METHOD setCirclePlane : BOOL //Return value = TRUE if executed succesful
VAR_INPUT
	X														: LREAL := 0.0;
	Y														: LREAL := 0.0;
	Z														: LREAL := 0.0;
	Q1														: LREAL := 0.0;
	Q2														: LREAL := 0.0;
	Q3														: LREAL := 0.0;
	Q4														: LREAL := 0.0;
	Q5														: LREAL := 0.0;
	Velo													: LREAL; 	// mm/s 
	AccurateStop											: BOOL := FALSE;
	Clockwise												: BOOL := TRUE;
	Plane													: E_NciGeoPlane := E_NciGeoPlaneXY;
	CenterX													: LREAL := 0.0;
	CenterY													: LREAL := 0.0;
	CenterZ													: LREAL := 0.0;
END_VAR
	(* NCI GeoCirclePlane schreiben									*)
	(*********************************************************)

(* Zielpos. in Tabelle schreiben ************************************************************)
	BlockCount 												:= BlockCount + 1;
	TblTemplate.GeoCirclePlane.nDisplayIndex := LastBlockNo := SEL(BlockNo = 0, BlockNo, TableNumber * OffsetFactorTblNumber + BlockCount);
	TblTemplate.GeoCirclePlane.fEndPosX						:= X;
	TblTemplate.GeoCirclePlane.fEndPosY						:= Y;
	TblTemplate.GeoCirclePlane.fEndPosZ						:= Z;
	TblTemplate.GeoCirclePlane.fEndPosQ1					:= Q1;
	TblTemplate.GeoCirclePlane.fEndPosQ2					:= Q2;
	TblTemplate.GeoCirclePlane.fEndPosQ3					:= Q3;
	TblTemplate.GeoCirclePlane.fEndPosQ4					:= Q4;
	TblTemplate.GeoCirclePlane.fEndPosQ5					:= Q5;
	TblTemplate.GeoCirclePlane.fVelo						:= Velo;
	TblTemplate.GeoCirclePlane.bAccurateStop				:= AccurateStop;
	TblTemplate.GeoCirclePlane.bClockwise					:= Clockwise;
	TblTemplate.GeoCirclePlane.nPlane						:= Plane;
	TblTemplate.GeoCirclePlane.fCenterX						:= CenterX;
	TblTemplate.GeoCirclePlane.fCenterY						:= CenterY;
	TblTemplate.GeoCirclePlane.fCenterZ						:= CenterZ;
                                                        	
	TblTemplate.InsertGeoCirclePlane(Table:= Table);    	
	Error													:= TblTemplate.Error;
	ErrorId													:= TblTemplate.ErrorId;
	ErrorText												:= TblTemplate.ErrorText;
	FilledRows												:= TblTemplate.FilledRows;

	SetCirclePlane											:= NOT Error;
(***************************************************************************)
END_METHOD

METHOD setCoordinateSystem : BOOL //Return value = TRUE if executed succesful
VAR_INPUT
	/// UCS ObjectID 
	ObjectId												: UDINT := 0;
END_VAR
(* NCI UserKos schreiben															*)
(************************************************************************************)

(* User Koordinatensystem schreiben ************************************************************)
	BlockCount 												:= BlockCount + 1;
	TblTemplate.SetCoordinateSystem.nDisplayIndex := LastBlockNo := SEL(BlockNo = 0, BlockNo, TableNumber * OffsetFactorTblNumber + BlockCount);
	TblTemplate.SetCoordinateSystem.nObjectId				:= ObjectId;

	TblTemplate.InsertSetCoordinateSystem(Table:= Table);
	Error													:= TblTemplate.Error;
	ErrorId													:= TblTemplate.ErrorId;
	ErrorText												:= TblTemplate.ErrorText;
	FilledRows												:= TblTemplate.FilledRows;
	
	SetCoordinateSystem										:= not Error;
(*************************************************************************************)
END_METHOD

METHOD setDynOverride : BOOL //Return value = TRUE if executed succesful
VAR_INPUT
	/// UCS ObjectID 
	Value													: lreal := 0; //0.0-100.0%
END_VAR
(* NCI Oevrride schreiben											*)
(********************************************************************)

(* insert override **************************************************)
	(* apapt override *)
	BlockCount 												:= BlockCount + 1;
	TblTemplate.DynOverride.nDisplayIndex := LastBlockNo 		:= SEL(BlockNo = 0, BlockNo, TableNumber * OffsetFactorTblNumber + BlockCount);
	TblTemplate.DynOverride.fDynOvr								:= 0.01 * Value;

	TblTemplate.InsertDynOverride(Table:= Table);
	Error													:= TblTemplate.Error;
	ErrorId													:= TblTemplate.ErrorId;
	ErrorText												:= TblTemplate.ErrorText;
	FilledRows												:= TblTemplate.FilledRows;
	
	SetDynOverride											:= not Error;
(*************************************************************************************)
END_METHOD

METHOD setGeoBezier3 : booL //Return value = TRUE if executed succesful
VAR_INPUT
     ControlPoint1X											: LREAL;
     ControlPoint1Y											: LREAL;
     ControlPoint1Z											: LREAL;
     ControlPoint2X											: LREAL;
     ControlPoint2Y											: LREAL;
     ControlPoint2Z											: LREAL;
     EndPosX												: LREAL;
     EndPosY												: LREAL;
     EndPosZ												: LREAL;
     EndPosQ1												: LREAL;
     EndPosQ2												: LREAL;
     EndPosQ3												: LREAL;
     EndPosQ4												: LREAL;
     EndPosQ5												: LREAL;
     Velo													: LREAL;
     AccurateStop											: BOOL; (* VeloEnd := 0 *)
END_VAR
	(* NCI SetGeoBezier3 schreiben						*)
	(*********************************************************)

(* Zielpos. in Tabelle schreiben ************************************************************)
	BlockCount 												:= BlockCount + 1;
	TblTemplate.GeoBezier3.nDisplayIndex := LastBlockNo := SEL(BlockNo = 0, BlockNo, TableNumber * OffsetFactorTblNumber + BlockCount);

    TblTemplate.GeoBezier3.fControlPoint1X					:= ControlPoint1X;
    TblTemplate.GeoBezier3.fControlPoint1Y					:= ControlPoint1Y;
    TblTemplate.GeoBezier3.fControlPoint1Z					:= ControlPoint1Z;
    TblTemplate.GeoBezier3.fControlPoint2X					:= ControlPoint2X;
    TblTemplate.GeoBezier3.fControlPoint2Y					:= ControlPoint2Y;
    TblTemplate.GeoBezier3.fControlPoint2Z					:= ControlPoint2Z;
    TblTemplate.GeoBezier3.fEndPosX							:= EndPosX;
    TblTemplate.GeoBezier3.fEndPosY							:= EndPosY;
    TblTemplate.GeoBezier3.fEndPosZ							:= EndPosZ;
    TblTemplate.GeoBezier3.fEndPosQ1						:= EndPosQ1;
    TblTemplate.GeoBezier3.fEndPosQ2						:= EndPosQ2;
    TblTemplate.GeoBezier3.fEndPosQ3						:= EndPosQ3;
    TblTemplate.GeoBezier3.fEndPosQ4						:= EndPosQ4;
    TblTemplate.GeoBezier3.fEndPosQ5						:= EndPosQ5;
    TblTemplate.GeoBezier3.fVelo							:= Velo;
    TblTemplate.GeoBezier3.bAccurateStop					:= AccurateStop  ;                            	
	
	TblTemplate.InsertGeoBezier3(Table:= Table);    	
	Error													:= TblTemplate.Error;
	ErrorId													:= TblTemplate.ErrorId;
	ErrorText												:= TblTemplate.ErrorText;
	FilledRows												:= TblTemplate.FilledRows;

	SetGeoBezier3											:= NOT Error;
(***************************************************************************)
END_METHOD

METHOD setGeoBezier5 : booL //Return value = TRUE if executed succesful
VAR_INPUT
     ControlPoint1X											: LREAL;
     ControlPoint1Y											: LREAL;
     ControlPoint1Z											: LREAL;
     ControlPoint2X											: LREAL;
     ControlPoint2Y											: LREAL;
     ControlPoint2Z											: LREAL;
     ControlPoint3X											: LREAL;
     ControlPoint3Y											: LREAL;
     ControlPoint3Z											: LREAL;
     ControlPoint4X											: LREAL;
     ControlPoint4Y											: LREAL;
     ControlPoint4Z											: LREAL;
     EndPosX												: LREAL;
     EndPosY												: LREAL;
     EndPosZ												: LREAL;
     EndPosQ1												: LREAL;
     EndPosQ2												: LREAL;
     EndPosQ3												: LREAL;
     EndPosQ4												: LREAL;
     EndPosQ5												: LREAL;
     Velo													: LREAL;
     AccurateStop											: BOOL; (* VeloEnd := 0 *)
END_VAR
	(* NCI SetGeoBezier5 schreiben						*)
	(*********************************************************)

(* Zielpos. in Tabelle schreiben ************************************************************)
	BlockCount 												:= BlockCount + 1;
	TblTemplate.GeoBezier5.nDisplayIndex := LastBlockNo := SEL(BlockNo = 0, BlockNo, TableNumber * OffsetFactorTblNumber + BlockCount);

    TblTemplate.GeoBezier5.fControlPoint1X					:= ControlPoint1X;
    TblTemplate.GeoBezier5.fControlPoint1Y					:= ControlPoint1Y;
    TblTemplate.GeoBezier5.fControlPoint1Z					:= ControlPoint1Z;
    TblTemplate.GeoBezier5.fControlPoint2X					:= ControlPoint2X;
    TblTemplate.GeoBezier5.fControlPoint2Y					:= ControlPoint2Y;
    TblTemplate.GeoBezier5.fControlPoint2Z					:= ControlPoint2Z;
    TblTemplate.GeoBezier5.fControlPoint3X					:= ControlPoint3X;
    TblTemplate.GeoBezier5.fControlPoint3Y					:= ControlPoint3Y;
    TblTemplate.GeoBezier5.fControlPoint3Z					:= ControlPoint3Z;
    TblTemplate.GeoBezier5.fControlPoint4X					:= ControlPoint4X;
    TblTemplate.GeoBezier5.fControlPoint4Y					:= ControlPoint4Y;
    TblTemplate.GeoBezier5.fControlPoint4Z					:= ControlPoint4Z;
    TblTemplate.GeoBezier5.fEndPosX							:= EndPosX;
    TblTemplate.GeoBezier5.fEndPosY							:= EndPosY;
    TblTemplate.GeoBezier5.fEndPosZ							:= EndPosZ;
    TblTemplate.GeoBezier5.fEndPosQ1						:= EndPosQ1;
    TblTemplate.GeoBezier5.fEndPosQ2						:= EndPosQ2;
    TblTemplate.GeoBezier5.fEndPosQ3						:= EndPosQ3;
    TblTemplate.GeoBezier5.fEndPosQ4						:= EndPosQ4;
    TblTemplate.GeoBezier5.fEndPosQ5						:= EndPosQ5;
    TblTemplate.GeoBezier5.fVelo							:= Velo;
    TblTemplate.GeoBezier5.bAccurateStop					:= AccurateStop  ;                            	
	
	TblTemplate.InsertGeoBezier5(Table:= Table);    	
	Error													:= TblTemplate.Error;
	ErrorId													:= TblTemplate.ErrorId;
	ErrorText												:= TblTemplate.ErrorText;
	FilledRows												:= TblTemplate.FilledRows;

	SetGeoBezier5											:= NOT Error;
(***************************************************************************)
END_METHOD

METHOD setGeoLine : BOOL //Return value = TRUE if executed succesful
VAR_INPUT
	X														: LREAL := 0.0;
	Y														: LREAL := 0.0;
	Z														: LREAL := 0.0;
	Q1														: LREAL := 0.0;
	Q2														: LREAL := 0.0;
	Q3														: LREAL := 0.0;
	Q4														: LREAL := 0.0;
	Q5														: LREAL := 0.0;
	Velo													: LREAL; 	// mm/s 
	AccurateStop											: BOOL := FALSE;
END_VAR
(* writing NCI GeoLine 									*)
(********************************************************)

(***************************************************************************)
	BlockCount 												:= BlockCount + 1;
	TblTemplate.GeoLine.nDisplayIndex := LastBlockNo 		:= SEL(BlockNo = 0, BlockNo, TableNumber * OffsetFactorTblNumber + BlockCount);
	TblTemplate.GeoLine.fEndPosX							:= X;
	TblTemplate.GeoLine.fEndPosY							:= Y;
	TblTemplate.GeoLine.fEndPosZ							:= Z;
	TblTemplate.GeoLine.fEndPosQ1							:= Q1 ;
	TblTemplate.GeoLine.fEndPosQ2							:= Q2;
	TblTemplate.GeoLine.fEndPosQ3							:= Q3;
	TblTemplate.GeoLine.fEndPosQ4							:= Q4;
	TblTemplate.GeoLine.fEndPosQ5							:= Q5;
	TblTemplate.GeoLine.fVelo								:= Velo;
	TblTemplate.GeoLine.bRapidTraverse						:= Velo = 0.0;
	TblTemplate.GeoLine.bAccurateStop						:= AccurateStop;
                                                        	
	TblTemplate.InsertGeoLine(Table:= Table);           	
	Error													:= TblTemplate.Error;
	ErrorId													:= TblTemplate.ErrorId;
	ErrorText												:= TblTemplate.ErrorText;
	FilledRows												:= TblTemplate.FilledRows;
	
	SetGeoLine												:= not Error;
(***************************************************************************)
END_METHOD

METHOD setGeoStart : BOOL //Return value = TRUE if executed succesful
VAR_INPUT
	X														: LREAL := 0.0;
	Y														: LREAL := 0.0;
	Z														: LREAL := 0.0;
	Q1														: LREAL := 0.0;
	Q2														: LREAL := 0.0;
	Q3														: LREAL := 0.0;
	Q4														: LREAL := 0.0;
	Q5														: LREAL := 0.0;
END_VAR
(* writing NCI GeoLine 									*)
(********************************************************)

(***************************************************************************)
	TblTemplate.GeoStart.fPosX								:= X;
	TblTemplate.GeoStart.fPosY								:= Y;
	TblTemplate.GeoStart.fPosZ								:= Z;
	TblTemplate.GeoStart.fPosQ1								:= Q1 ;
	TblTemplate.GeoStart.fPosQ2								:= Q2;
	TblTemplate.GeoStart.fPosQ3								:= Q3;
	TblTemplate.GeoStart.fPosQ4								:= Q4;
	TblTemplate.GeoStart.fPosQ5								:= Q5;
                                                        	
	TblTemplate.InsertGeoStart(Table:= Table);           	
	Error													:= TblTemplate.Error;
	ErrorId													:= TblTemplate.ErrorId;
	ErrorText												:= TblTemplate.ErrorText;
	FilledRows												:= TblTemplate.FilledRows;
	
	SetGeoStart												:= not Error;
(***************************************************************************)
END_METHOD

METHOD setHParam : booL //Return value = TRUE if executed succesful
VAR_INPUT
	HParam													: UDINT;
END_VAR
(* 														*)
(********************************************************)

(*************************************************************************************)
	BlockCount 												:= BlockCount + 1;
	TblTemplate.HParam.nDisplayIndex := LastBlockNo 		:= SEL(BlockNo = 0, BlockNo,  TableNumber * OffsetFactorTblNumber + BlockCount);
	TblTemplate.HParam.nHParam								:= HParam;
                                                        	
	TblTemplate.InsertHParam(Table:= Table);          	
	Error													:= TblTemplate.Error;
	ErrorId													:= TblTemplate.ErrorId;
	ErrorText												:= TblTemplate.ErrorText;
	FilledRows												:= TblTemplate.FilledRows;
	
	SetHParam												:= NOT Error;
(*************************************************************************************)
END_METHOD

METHOD setPathDynamics : BOOL //Return value = TRUE if executed succesful
VAR_INPUT
	Acc,Dec,Jerk											:	LREAL;
END_VAR
	(* NCI SetPathDynamics schreiben						*)
	(*********************************************************)

(* Zielpos. in Tabelle schreiben ************************************************************)
	BlockCount 												:= BlockCount + 1;
	TblTemplate.PathDynamics.nDisplayIndex := LastBlockNo := SEL(BlockNo = 0, BlockNo, TableNumber * OffsetFactorTblNumber + BlockCount);

	TblTemplate.PathDynamics.fDec							:= Dec;
	TblTemplate.PathDynamics.fJerk							:= Jerk;
	TblTemplate.PathDynamics.fAcc							:= Acc;
                                                        	
	TblTemplate.InsertPathDynamics(Table:= Table);    	
	Error													:= TblTemplate.Error;
	ErrorId													:= TblTemplate.ErrorId;
	ErrorText												:= TblTemplate.ErrorText;
	FilledRows												:= TblTemplate.FilledRows;

	SetPathDynamics											:= NOT Error;
(***************************************************************************)
END_METHOD

METHOD setSParam : bool //Return value = TRUE if executed succesful
VAR_INPUT
	SParam													: UINT;
END_VAR
(* 														*)
(********************************************************)

(*************************************************************************************)
	BlockCount 												:= BlockCount + 1;
	TblTemplate.SParam.nDisplayIndex := LastBlockNo 		:= SEL(BlockNo = 0, BlockNo,  TableNumber * OffsetFactorTblNumber + BlockCount);
	TblTemplate.SParam.nSParam								:= SParam;
                                                        	
	TblTemplate.InsertSParam(Table:= Table);          	
	Error													:= TblTemplate.Error;
	ErrorId													:= TblTemplate.ErrorId;
	ErrorText												:= TblTemplate.ErrorText;
	FilledRows												:= TblTemplate.FilledRows;
	
	SetSParam												:= NOT Error;
(*************************************************************************************)
END_METHOD

METHOD setTangFollowingDesc : booL //Return value = TRUE if executed succesful
VAR_INPUT
    TangOn													: BOOL;
    TangAxis												: E_NciAxesInGroup;  
    PathAxis1												: E_NciAxesInGroup; 
    PathAxis2												: E_NciAxesInGroup; 
    Offset													: LREAL; 
    CriticalAngle1											: LREAL;
    TfBehavior												: E_TangentialFollowingBehavior; 
END_VAR
	(* NCI SetTangFollowingDesc schreiben						*)
	(*********************************************************)

(* Zielpos. in Tabelle schreiben ************************************************************)
	BlockCount 												:= BlockCount + 1;
	LastBlockNo 											:= SEL(BlockNo = 0, BlockNo, TableNumber * OffsetFactorTblNumber + BlockCount);

    TblTemplate.TangentialFollowingDesc.bTangOn				:= TangOn;
    TblTemplate.TangentialFollowingDesc.nTangAxis			:= TangAxis;
    TblTemplate.TangentialFollowingDesc.nPathAxis1			:= PathAxis1;
    TblTemplate.TangentialFollowingDesc.nPathAxis2			:= PathAxis2;
    TblTemplate.TangentialFollowingDesc.fOffset				:= Offset;
    TblTemplate.TangentialFollowingDesc.fCriticalAngle1		:= CriticalAngle1;
    TblTemplate.TangentialFollowingDesc.nTfBehavior			:= TfBehavior;
                       	
	TblTemplate.InsertTangFollowingDesc(Table:= Table);    	
	Error													:= TblTemplate.Error;
	ErrorId													:= TblTemplate.ErrorId;
	ErrorText												:= TblTemplate.ErrorText;
	FilledRows												:= TblTemplate.FilledRows;

	SetTangFollowingDesc									:= NOT Error;
(***************************************************************************)
END_METHOD

METHOD setTParam : bool //Return value = TRUE if executed succesful
VAR_INPUT
	TParam													: UINT;
END_VAR
(* 														*)
(********************************************************)

(*************************************************************************************)
	BlockCount 												:= BlockCount + 1;
	TblTemplate.TParam.nDisplayIndex := LastBlockNo 		:= SEL(BlockNo = 0, BlockNo,  TableNumber * OffsetFactorTblNumber + BlockCount);
	TblTemplate.TParam.nTParam								:= TParam;
                                                        	
	TblTemplate.InsertTParam(Table:= Table);          	
	Error													:= TblTemplate.Error;
	ErrorId													:= TblTemplate.ErrorId;
	ErrorText												:= TblTemplate.ErrorText;
	FilledRows												:= TblTemplate.FilledRows;
	
	SetTParam												:= NOT Error;
(**************************************************************************)
END_METHOD

METHOD setVertexSmoothing : BOOL //Return value = TRUE if executed succesful
VAR_INPUT
	Radius													: LREAL := 0.0;
	VertSmType												: UDINT := 5;
	VertSmSubType											: UDINT := 3;
END_VAR
(* writing NCI Vertex smoothing 								*)
(****************************************************************)

(* writing into table	*****************************************)
	BlockCount 												:= BlockCount + 1;
	TblTemplate.VertexSmoothing.nDisplayIndex := LastBlockNo := SEL(BlockNo = 0, BlockNo, TableNumber * OffsetFactorTblNumber + BlockCount);
	TblTemplate.VertexSmoothing.nType						:= VertSmType;
	TblTemplate.VertexSmoothing.nSubtype					:= VertSmSubtype; (* 	1: constant radius tolerance
																					2: distance between Abstand intersectoin point and peal point
																					3: adaptiv raidus tolerance
																					*)
	TblTemplate.VertexSmoothing.fRadius						:= Radius; (* mm *)

	TblTemplate.InsertVertexSmoothing(Table:= Table);
	Error													:= TblTemplate.Error;
	ErrorId													:= TblTemplate.ErrorId;
	ErrorText												:= TblTemplate.ErrorText;
	FilledRows												:= TblTemplate.FilledRows;
	SetVertexSmoothing										:= not Error;
(*************************************************************************************)
END_METHOD

END_FUNCTION_BLOCK

// ---- POUs/Motion/TF511x-KIN/KinChannel.TcPOU
FUNCTION_BLOCK KinChannel EXTENDS KIN_REF
VAR_INPUT
	Admin													:	KinAdmin;
END_VAR
VAR_OUTPUT
END_VAR
VAR
END_VAR

(* Kinematic Ctrl 										*)
(********************************************************)

(* work IO ********************************************************************)
(*	IO(); *)
	
(****************************************************************************)
(* Kinematic group control													*)
(****************************************************************************)
	Admin(
		ResetTrig			:= ,
		Enable			:= ,
		Override		:= ,
		ItpChannelId	:= ,
		AxesList		:= ,
		rKINRef			:= THIS^,
		Busy			=> ,
		Done			=> ,
		Error			=> ,
		ErrorId			=> );
(****************************************************************************)

END_FUNCTION_BLOCK

// ---- POUs/Motion/TF50xx-NC/02_Options/Coupling/AxCamming.TcPOU
{attribute 'no_check'}
//Nc-axis camming (cam tabel) control
//based on Tc2_MC2_Camming library
FUNCTION_BLOCK AxCamming EXTENDS AxFbBase
VAR_OUTPUT CONSTANT
	FNC_CAM_OUT												:	INT := 0;
	FNC_CAM_IN												:	INT := 1;
END_VAR                     								
VAR_INPUT                   								
	Fnc														:	INT (FNC_CAM_OUT..FNC_CAM_IN) := FNC_CAM_OUT;
	MasterOffset											:	LREAL		:= 0.0;
	SlaveOffset												:	LREAL 	:= 0.0;
	MasterScaling											:	LREAL 	:= 1.0;
	SlaveScaling											:	LREAL 	:= 1.0;
	MasterScalingMode										:	MC_CamScalingMode := MC_CAMSCALING_USERDEFINED;
	SlaveScalingMode										:	MC_CamScalingMode := MC_CAMSCALING_USERDEFINED;
	StartMode  												:	MC_StartMode := MC_STARTMODE_ABSOLUTE; 	(* StartMode determines whether the cam plate position is interpreted absolute OR relative TO the coupling position.StartMode can be relative OR absolute FOR master (X coordinate) AND slave (Y coordinate). *)
	TableID  												:	MC_CAM_ID; 		(*ID der Kurvenscheibe mit der gekoppelt wird *)
	ActivationMode											:	MC_CamActivationMode := MC_CAMACTIVATION_INSTANTANEOUS;
	ActivationPosition										:	LREAL := 0.0;
	InterpolationType										:	MC_InterpolationType := MC_INTERPOLATIONTYPE_LINEAR;

	rMasterAxis												:	REFERENCE TO AXIS_REF := 0;
END_VAR
VAR_IN_OUT
END_VAR
VAR_OUTPUT
END_VAR
VAR
(* cache *******************************************************************)
	MemFnc													:	INT := -1;

(* timer *)

(* trigger *)

(* MC-function-block instances *********************************************)
	MC_CamIn												:	MC_CamIn;
	MC_CamOut												:	MC_CamOut;

END_VAR

	(* NC axis cam table control														*)
	(************************************************************************************)

(* Execute ***************************************************************************************)
	rtExecute(CLK := Execute);
	IF rtExecute.Q
		AND MemFnc < 0
	THEN
		MemFnc 												:= Fnc ;
		Busy												:= TRUE;
		Done												:= FALSE;
		Error												:= FALSE;
		ErrorID												:= 0;
		CmdAborted											:= FALSE;
		ErrorText											:= '';
	END_IF

(* Call Method ***********************************************************************************)
	CASE MemFnc OF
	FNC_CAM_OUT:
		CamOut(Execute);

	FNC_CAM_IN:
		CamIn(Execute);

	-1:
		IF NOT Execute
		THEN
			Busy											:= FALSE;
			Done											:= FALSE;
			Error											:= FALSE;
			ErrorID											:= 0;
			CmdAborted										:= FALSE;
			ErrorText										:= '';
		END_IF                              				
	ELSE                                    				
		Busy												:= FALSE;
		Done												:= FALSE;
		Error												:= Execute;
		ErrorID												:= E_AdsErr.DEVICE_INVALIDPARM;
		CmdAborted											:= FALSE;
		ErrorText											:= CONCAT('invalid parameter value(s) Fnc no: ' , INT_TO_STRING(MemFnc));
	END_CASE

(*************************************************************************************************)

METHOD PUBLIC camIn : BOOL //Return value = TRUE if busy
//required parameter
//rAxis
//rMasterAxis
//MasterOffset
//SlaveOffset
//MasterScaling
//SlaveScaling
//StartMode
//CamTableID
//Options
VAR_INPUT
	Execute													:	BOOL;
END_VAR
MemFnc														:= FNC_CAM_IN;
THIS^.Execute												:= Execute;
	
IF NOT __ISVALIDREF(rAxis) 
THEN
	Busy													:= NOT Error;
	Error													:= TRUE;
	ErrorId													:= E_AdsErr.DEVICE_INVALIDPARM;
	CmdAborted												:= FALSE;
	Done													:= FALSE;
	Active													:= FALSE;
	ErrorText												:= 'Reference rAxis invalid (0)';
	MemFnc													:= SEL(Execute , -1 ,MemFnc); 
	RETURN;
ELSIF NOT __ISVALIDREF(rMasterAxis)
THEN
	Busy													:= NOT Error;
	Error													:= TRUE;
	ErrorId													:= E_AdsErr.DEVICE_INVALIDPARM;
	CmdAborted												:= FALSE;
	Done													:= FALSE;
	ErrorText												:= 'Reference rMasterAxis invalid (0)';
	MemFnc													:= SEL(Execute , -1 ,MemFnc); 
	RETURN;
END_IF
	MC_CamIn.Options.ActivationMode							:= ActivationMode;
	MC_CamIn.Options.ActivationPosition						:= ActivationPosition;
	MC_CamIn.Options.MasterScalingMode						:= MasterScalingMode;
	MC_CamIn.Options.SlaveScalingMode						:= SlaveScalingMode;
	MC_CamIn.Options.InterpolationType						:= InterpolationType;

	MC_CamIn(
		Execute			:= Execute,
		MasterOffset	:= MasterOffset,
		SlaveOffset		:= SlaveOffset,
		MasterScaling	:= MasterScaling,
		SlaveScaling	:= SlaveScaling,
		StartMode		:= StartMode,
		CamTableID		:= TableID,
		BufferMode		:= ,
		Options			:= ,
		Master			:= rMasterAxis,
		Slave			:= rAxis,
		InSync			=> Done,
		Busy			=> Busy,
		Active			=> Active,
		CommandAborted	=> CmdAborted,
		Error			=> Error,
		ErrorID			=> ErrorID);

	IF Error THEN
		LastErrorId											:= ErrorId;
		ErrorText 											:= CONCAT('MC_CamIn ID:' , UDINT_TO_STRING(ErrorId));
	ELSE                    								
		ErrorText 											:= '';
	END_IF
	IF NOT MC_CamIn.Execute AND NOT Busy
	THEN
		MemFnc												:= -1  ;
	END_IF
END_METHOD

METHOD PUBLIC camOut : BOOL //Return value = TRUE if busy
//required parameter
//rAxis
VAR_INPUT
	Execute													:	BOOL;
END_VAR
	MemFnc													:= FNC_CAM_OUT;
	THIS^.Execute											:= Execute;
	
IF NOT __ISVALIDREF(rAxis) 
THEN
	Busy													:= NOT Error;
	Error													:= TRUE;
	ErrorId													:= E_AdsErr.DEVICE_INVALIDPARM;
	CmdAborted												:= FALSE;
	Done													:= FALSE;
	Active													:= FALSE;
	ErrorText												:= 'Reference rAxis invalid (0)';
	MemFnc													:= SEL(Execute , -1 ,MemFnc); 
	RETURN;
END_IF
	
	MC_CamOut(
		Execute	:= Execute,
		Options	:= ,
		Slave	:= rAxis,
		Done	=> Done,
		Busy	=> Busy,
		Error	=> Error,
		ErrorID	=> ErrorID);

	Active													:= Busy;
	CmdAborted												:= FALSE;

	IF Error THEN
		LastErrorId											:= ErrorId;
		ErrorText 											:= CONCAT('MC_CamOut ID:' , UDINT_TO_STRING(ErrorId));
	ELSE
		ErrorText 											:= '';
	END_IF

	IF NOT Execute AND NOT Busy
	THEN
		MemFnc												:= -1;
	END_IF
END_METHOD

END_FUNCTION_BLOCK

// ---- POUs/Motion/TF50xx-NC/02_Options/Motion/AxMoveSinus.TcPOU
{attribute 'pack_mode' := '4'}
FUNCTION_BLOCK AxMoveSinus EXTENDS FbBase
VAR_INPUT
	Frequence												: LREAL := 0.0; //Hz
	SinusVeloAmplitude										: LREAL := 0.0; //mm/s
	DrivingTime												: TIME := T#0MS; //s
END_VAR
VAR_IN_OUT
	Axis													: AXIS_REF;
END_VAR
VAR_OUTPUT
	Active													: booL := FALSE;
	CommandAborted											: BOOL := FALSE;
END_VAR
VAR //Sinus Oscillation Sequence
(* 
- used as single sinus oscillation (sinus generator)
- used as sinus oscillation sequence (e.g. for bode plot) NEW 
UINT32 ENUM 1 				start type (fixed to start type 1 yet) 
UINT32 Reserved			
REAL64 e.g. mm/s > 0.0 		base amplitude (e.g. 2.5 mm/s) 
REAL64 Hz [0.0 .... 10.0] 	base frequency (e.g. 1.953125 Hz) 
REAL64 e.g. mm/s ≥ 0.0 		start amplitude at begin (e.g. 0.0 mm/s) 
REAL64 e.g. mm/REV > 0.0 	feed constant motor (per motor turn) (e.g. 10.0 mm/REV) 
REAL64 Hz ≥ 1.0 			frequency range: start frequency (e.g. 20.0 Hz) 
REAL64 Hz ≤ 1/(2*dT) 		frequency range: stop frequency (e.g. 500.0 Hz) 
REAL64 s > 0.0 				step duration (e.g. 2.048s) 
UINT32 1 [1 ... 200] 		number of measurements (step cycles) (e.g. 20) 
UINT32 1   					number of parallel measurements (e.g. 1)   not used yet! 
=72
*)   
	StartType												:	UDINT := TO_UDINT(Tc2_MC2._E_TCNC_StartPosType.TCNC_START_ABSOLUTE);
	Reserved												:	UDINT := 0;	
	BaseAmplitude											:	LREAL := 2.5;
	BaseFrequency											:	LREAL := 1.953125;
	StartAmplitude											:	LREAL := 0.0;
	FeedConstantMotor										:	LREAL := 10.0;
	FreqRangeStartFreq										:	LREAL := 0.0;
	FreqRangeStopFreq										:	LREAL := 500.0;								
	StepDuration											:	LREAL := 0.0;
	NumOfMeasurements										:	UDINT  := 0; //StepCount
	NumOfParallelMeasurements								:	UDINT  := 1;	
END_VAR
VAR
(* Internal memory **********************************************************************)
	LastErrorID												:	UDINT;
	StartCmdNo												: WORD;
	
(* Timer ********************************************************************************)                 	
	tonTimeout												:	TON;

(* Trigger ******************************************************************************)

(* FB instances *************************************************************************)
	Write_ADS												: ADSWRITE  := (NetId := '', Port := AMSPORT_R0_NCSAF, IdxGrp := 16#4200 + 0, IdxOffs := 16#33, LEN := 72, TmOut := DEFAULT_ADS_TIMEOUT);

(* Dummys *******************************************************************************)

END_VAR


(* Sinus Oscillation Sequence *************************************************************************************)
rtExecute(CLK := Execute);
CASE State OF
0://Wait for execute signal to change state to true
	IF NOT Execute OR rtExecute.Q	
	THEN
		Write_Ads(WRITE := FALSE);
		tonTimeout(IN := FALSE);
		FreqRangeStartFreq									:= Frequence;
		StartAmplitude										:= SinusVeloAmplitude;
		StepDuration										:= TO_LREAL(DrivingTime) * 0.001; //time ms to lreal s
		Busy												:= rtExecute.Q;
		CommandAborted										:= FALSE;
		Active												:= FALSE;
		Done 												:= FALSE;
		Error												:= FALSE;
		ErrorID												:= 0;
		StartCmdNo											:= Axis.NcToPlc.CmdNo;

		Write_ADS( //See also declaration
			IdxGrp	:=	16#4200+Axis.NcToPlc.AxisId,
			SrcAddr	:=ADR(StartType), 
			Write 	:= rtExecute.Q);
		
		state												:= SEL(Write_ADS.Write, 0, state + 1);
	
	END_IF

1://Read original parameters for position lag monitoring
	Write_ADS(SrcAddr	:=ADR(StartType)); 
	IF NOT Write_ADS.BUSY 
	THEN
		IF Write_ADS.ERR 
		THEN
			LastErrorId										:= Write_ADS.ERRID;	
			BUSY 											:= FALSE;
			Error											:= TRUE;
			ErrorId											:= LastErrorId;
			State											:= 0;
		ELSE				
			Active 											:= F_AxisHasJob(Axis.NcToPlc.StateDWord) AND StartCmdNo <> Axis.NcToPlc.CmdNo;	
			state											:= state + 1;
		END_IF
		Write_ADS(Write := FALSE);
	END_IF

2: //Wait for command done
	IF F_AxisHasJob(Axis.NcToPlc.StateDWord) AND StartCmdNo <> Axis.NcToPlc.CmdNo
	THEN
		Active												:= TRUE;
	ELSIF F_AxisInErrorState(Axis.NcToPlc.StateDWord) 
	THEN
		Active												:= FALSE;
		Busy												:= FALSE;
		(* axis error came up before this command has been started *)
		Error 												:= TRUE;
		ErrorID 											:= AXIS.NcToPlc.ErrorCode;
		LastErrorId											:= ErrorId;
		state												:= 0;
		
	ELSIF F_AxisIsCoupled(Axis.NcToPlc.CoupleState) 
		OR F_AxisHasBeenStopped(Axis.NcToPlc.StateDWord) 
	THEN
		(* if axis is coupled during motion (FlyingSaw) all commands are aborted *)
		Active												:= FALSE;
		Busy												:= FALSE;
		CommandAborted 										:= TRUE;
		state												:= 0;																																     	

	ELSIF Active
	THEN //No longer active
		Active												:= FALSE;
		Busy												:= FALSE;
		Done												:= TRUE;
		state												:= 0;		
	ELSE 	
		tonTimeOut(In := TRUE, PT := T#100MS);
		IF tonTimeOut.Q
		THEN //Command not responded
			Busy											:= FALSE;
			Error 											:= TRUE;
			ErrorID 										:= MC_ERROR_STATE_FEEDBACK_TIMEOUT;
			state											:= 0;				
		END_IF			
	END_IF
END_CASE
(********************************************************************************************)

END_FUNCTION_BLOCK

// ---- POUs/Motion/TF50xx-NC/02_Options/Motion/AxHomingOnBlock.TcPOU
{attribute 'no_check'}
//Nc-axis homing on block sequence control for CoE drive 
//based on Tc2_MC2 library
FUNCTION_BLOCK AxHomingOnBlock EXTENDS FbBase
VAR CONSTANT	
	DEVICE_TYPE_PROFILE_DS402								:	UDINT := 5001;
	DEVICE_TYPE_PROFILE_MDP									:	UDINT := 131474;	
END_VAR
VAR_INPUT
	Position												: LREAL := DEFAULT_HOME_POSITION;//Used as homepos if value is <> DEFAULT_HOME_POSITION
	Direction												: MC_Direction := MC_Negative_Direction; //Homing direction
	Velocity												: LREAL := 0.0; //0.0 = Default NC valuse are used, else "Velocity" is used for both movements, into block direction and retraction
	Acceleration											: LREAL := 0.0; //0.0 = Default dynamics are used
	Deceleration											: LREAL := 0.0; //0.0 = Default dynamics are used
	Offset													: LREAL := 2.0; //Offset to release block
	LagTolerance											: LREAL	:= 0.5; //Lag error tolerance to detect axis on block
	MaxTorque												: LREAL	:= 50.0;//Max torque during homing towards block and retartion
	DrvChannel												: BYTE	:= 0; //Drive channel 0 or 1 
END_VAR
VAR_IN_OUT
	Axis													: AXIS_REF;
END_VAR
VAR_OUTPUT
	DriveProfileIsDS402										:	BOOL;							
END_VAR
VAR
(* Internal memory **********************************************************************)
	LastErrorState											: INT ; //Last error state for debugging
	LastErrorId												: UDINT;
	MemError												: BOOL;
	MemBlockPos												: LREAL;
	VelocityTowardsBlock									: LREAL;
	VelocityOffBlock										: LREAL;
	// Parameter storage for returning values to original after running the procedure.
	Param_DeviceType										: UDINT;
	Param_MotionMonitoring									: BYTE;
	Param_LagMonitoring										: BYTE;
	Param_SoftMaxMonitoring									: BYTE;
	Param_SoftMinMonitoring									: BYTE;	                        	
	Param_MaxTorque											: UINT;
	Param_MaxTorqueRead										: BOOL;
	Param_CalibrationValue									: LREAL;
	
(* Timer ********************************************************************************)                 	

(* Trigger ******************************************************************************)

(* FB instances *************************************************************************)
	Read_ADS												: ADSREAD := (TmOut := DEFAULT_ADS_TIMEOUT);
	Write_ADS												: ADSWRITE  := (TmOut := DEFAULT_ADS_TIMEOUT);
	MC_Home													: MC_Home;
	Mc_Halt													: MC_Halt;
	MC_Velocity												: MC_MoveVelocity;
	MC_Absolute												: MC_MoveAbsolute;
	CoEWrite												: FB_CoEWrite;
	CoERead													: FB_CoERead;
(* Dummys *******************************************************************************)
	uiValue													: UINT; //Temporary use for reading BOOL
END_VAR

	(* Homing on block function																		*)
	(*																								*)
	(* V1.0 2016/02/15 ABarrett																		*)
	(************************************************************************************************)
	
(* Sequence *************************************************************************************)
rtExecute(CLK := Execute);
CASE State OF
0://Wait for execute signal to change state to true
	IF NOT Execute OR rtExecute.Q	
	THEN
		Read_ADS(Read := FALSE);	Write_Ads(Write := FALSE);
		CoEWrite(Execute := FALSE,axis  := axis); CoERead(Execute := FALSE,axis  := axis);										
		MC_Home(Execute := FALSE,Axis := Axis);
		MC_Halt(Execute := FALSE,Axis := Axis);
		MC_Velocity(Execute := FALSE,Axis := Axis);
		MC_Absolute(Execute := FALSE,Axis := Axis);	
		Param_MotionMonitoring								:= 0;
		Param_LagMonitoring									:= 0;
		Param_SoftMaxMonitoring								:= 0;
		Param_SoftMinMonitoring								:= 0;
	
		Busy												:= rtExecute.Q;
		Done 												:= FALSE;
		Error												:= FALSE;
		ErrorID												:= 0;
		MemError											:= 0;
		state												:= SEL(rtExecute.Q, 0, 100);
	
	END_IF

(* Read original parameters for position lag monitoring, limit switches, max torque....... ************************************)
100:
	(* Read device type from drive *)
	CoERead( 
		NetId			:= '', 
		Index			:= 16#1000,
		SubIndex		:= 0, 
		pDstBuf			:= ADR(Param_DeviceType), 
		BufLen			:= SIZEOF(Param_DeviceType), 
		Execute			:= TRUE, 
		Axis			:= Axis );
	IF NOT CoERead.BUSY
	THEN
		IF CoERead.Error
		THEN
			MemError										:= TRUE;
			LastErrorState									:= state;
			LastErrorId										:= CoERead.AdsErrId;//or CANopenErrId;				
			State											:= 900;
		ELSE
			DriveProfileIsDS402								:= Param_DeviceType = DEVICE_TYPE_PROFILE_DS402; 
			CoERead(Execute := FALSE, Axis := Axis);	
			state											:= State + 1;
		END_IF		
	END_IF

101:
	Read_ADS(NetId:= '' , Port:=500, IdxGrp:=16#4000+Axis.NcToPlc.AxisId, IDxOffs:=16#11,
				LEN:=SIZEOF(uiValue), DestAddr:=ADR(uiValue), Read := TRUE );
	IF NOT Read_ADS.BUSY 
	THEN
		IF Read_Ads.ERR
		THEN
			MemError										:= TRUE;
			LastErrorState									:= state;
			LastErrorId										:= Read_Ads.ERRID;				
			State											:= 900;
		ELSE                                            	
			Param_MotionMonitoring.0						:= TRUE;                                    	
			Param_MotionMonitoring.1						:= TO_BOOL(uiValue);
			state											:= state + 1;
		END_IF
		Read_ADS(Read := FALSE);						
	END_IF
	
102:
	Read_ADS(NetId:= '' , Port:=500, IdxGrp:=16#6000+Axis.NcToPlc.AxisId, IDxOffs:=16#10,
				LEN:=SIZEOF(uiValue), DestAddr:=ADR(uiValue), Read := TRUE );
	IF NOT Read_ADS.BUSY 
	THEN
		IF Read_Ads.ERR
		THEN
			MemError										:= TRUE;
			LastErrorState									:= state;
			LastErrorId										:= Read_Ads.ERRID;				
			State											:= 900;
		ELSE                                            	
			Param_LagMonitoring.0							:= TRUE;                                    	
			Param_LagMonitoring.1							:= TO_BOOL(uiValue);
			state											:= state + 1;
		END_IF
		Read_ADS(Read := FALSE);						
	END_IF		
		
103:
	Read_ADS(NetId:= '' , Port:=500, IdxGrp:=16#5000+Axis.NcToPlc.AxisId, IDxOffs:=16#C,
				LEN:=SIZEOF(uiValue), DestAddr:=ADR(uiValue), Read := TRUE );
	IF NOT Read_ADS.BUSY 
	THEN
		IF Read_Ads.ERR
		THEN
			MemError										:= TRUE;
			LastErrorState									:= state;
			LastErrorId										:= Read_Ads.ERRID;				
			State											:= 900;
		ELSE                                            	
			Param_SoftMaxMonitoring.0						:= TRUE;                                    	
			Param_SoftMaxMonitoring.1						:= TO_BOOL(uiValue);
			state											:= state + 1;
		END_IF
		Read_ADS(Read := FALSE);						
	END_IF		
	
104:
	Read_ADS(NetId:= '' , Port:=500, IdxGrp:=16#5000+Axis.NcToPlc.AxisId, IDxOffs:=16#B,
				LEN:=SIZEOF(uiValue), DestAddr:=ADR(uiValue), Read := TRUE );
	IF NOT Read_ADS.BUSY 
	THEN
		IF Read_Ads.ERR
		THEN
			MemError										:= TRUE;
			LastErrorState									:= state;
			LastErrorId										:= Read_Ads.ERRID;				
			State											:= 900;
		ELSE                                            	
			Param_SoftMinMonitoring.0						:= TRUE;                                    	
			Param_SoftMinMonitoring.1						:= TO_BOOL(uiValue);
			state											:= State + 1;
		END_IF
		Read_ADS(Read := FALSE);						
	END_IF	

105:
	Read_ADS(NetId:= '' , Port:=500, IdxGrp:=16#5000+Axis.NcToPlc.AxisId, IDxOffs:=16#103,
				LEN:=SIZEOF(Param_CalibrationValue), DestAddr:=ADR(Param_CalibrationValue), Read := TRUE );
	IF NOT Read_ADS.BUSY 
	THEN
		IF Read_Ads.ERR
		THEN
			MemError										:= TRUE;
			LastErrorState									:= state;
			LastErrorId										:= Read_Ads.ERRID;				
			State											:= 900;
		ELSE                                            	
			state											:= State + 1;
		END_IF
		Read_ADS(Read := FALSE);						
	END_IF			
	
106://Read velocity to use towards block
	IF Velocity = 0.0
	THEN //Only read values if FB parameter is 0.0
		Read_ADS(NetId:= '' , Port:=500, IdxGrp:=16#4000+Axis.NcToPlc.AxisId, IDxOffs:=16#6,
					LEN:=SIZEOF(VelocityTowardsBlock), DestAddr:=ADR(VelocityTowardsBlock), Read := TRUE );
		IF NOT Read_ADS.BUSY 
		THEN
			IF Read_Ads.ERR
			THEN
				MemError									:= TRUE;
				LastErrorState								:= state;
				LastErrorId									:= Read_Ads.ERRID;				
				State										:= 900;
			ELSE                                            
				state										:= State + 1;
			END_IF                                          
			Read_ADS(Read := FALSE);						
		END_IF                                              
	ELSE	                                                
		VelocityTowardsBlock								:= Velocity;
		VelocityOffBlock									:= Velocity;
		state												:= 108;	//Skip this and next state
	END_IF
	
107://Read velocity to use away from block to home position
	Read_ADS(NetId:= '' , Port:=500, IdxGrp:=16#4000+Axis.NcToPlc.AxisId, IDxOffs:=16#7,
				LEN:=SIZEOF(VelocityOffBlock), DestAddr:=ADR(VelocityOffBlock), Read := TRUE );
	IF NOT Read_ADS.BUSY 
	THEN
		IF Read_Ads.ERR
		THEN
			MemError										:= TRUE;
			LastErrorState									:= state;
			LastErrorId										:= Read_Ads.ERRID;				
			State											:= 900;
		ELSE                                            	
			state											:= State + 1;
		END_IF
		Read_ADS(Read := FALSE);						
	END_IF	
		
108://Read CoE value for max torque
	IF DrvChannel = 1
	THEN
		CoERead.Index										:= SEL(DriveProfileIsDS402, 16#7110 , 	16#6872); 
		CoERead.SubIndex									:= SEL(DriveProfileIsDS402, 16#B  , 	16#0);
	ELSE //Channel 0
		CoERead.Index										:= SEL(DriveProfileIsDS402, 16#7010 , 	16#6072);
		CoERead.SubIndex									:= SEL(DriveProfileIsDS402, 16#B  , 	16#0);
 	END_IF 
	
	CoERead( 
		NetId			:= '', 
		Index			:= , //See above 
		SubIndex		:= , //See above 
		pDstBuf			:= ADR(uiValue), 
		BufLen			:= SIZEOF(uiValue), //2,
		Execute			:= TRUE, 
		Axis			:= Axis );
	IF NOT CoERead.BUSY
	THEN
		IF CoERead.Error
		THEN
			MemError										:= TRUE;
			LastErrorState									:= state;
			LastErrorId										:= CoERead.AdsErrId;//or CANopenErrId;				
			State											:= 900;
		ELSE
			Param_MaxTorqueRead								:= TRUE;
			Param_MaxTorque									:= uiValue;
			CoERead(Execute := FALSE, Axis := Axis);	
			state											:= 200;
		END_IF		
	END_IF
	
	
(* Write all parameters to needed settings *********************************************************)
200:
	uiValue													:= TO_UINT(FALSE);
	Write_ADS(NetId:= '' , Port:=500, IdxGrp:=16#4000+Axis.NcToPlc.AxisId, IDxOffs:=16#11,
				LEN:=SIZEOF(uiValue), SrcAddr:=ADR(uiValue), Write := TRUE );
	IF NOT Write_ADS.BUSY 
	THEN
		IF Write_ADS.ERR
		THEN
			MemError										:= TRUE;
			LastErrorState									:= state;
			LastErrorId										:= Read_Ads.ERRID;				
			State											:= 600; //Jump to state 600 to restore old entrys
		ELSE
			state											:= state + 1;
		END_IF
		Write_ADS(Write := FALSE);						
	END_IF

201:
	uiValue													:= TO_UINT(FALSE);
	Write_ADS(NetId:= '' , Port:=500, IdxGrp:=16#6000+Axis.NcToPlc.AxisId, IDxOffs:=16#10,
				LEN:=SIZEOF(uiValue), SrcAddr:=ADR(uiValue), Write := TRUE );
	IF NOT Write_ADS.BUSY 
	THEN
		IF Write_ADS.ERR
		THEN
			MemError										:= TRUE;
			LastErrorState									:= state;
			LastErrorId										:= Read_Ads.ERRID;				
			State											:= 600; //Jump to state 600 to restore old entrys
		ELSE
			state											:= state + 1;
		END_IF
		Write_ADS(Write := FALSE);						
	END_IF

202:	
	uiValue													:= TO_UINT(FALSE);
	Write_ADS(NetId:= '' , Port:=500, IdxGrp:=16#5000+Axis.NcToPlc.AxisId, IDxOffs:=16#C,
					LEN:=SIZEOF(uiValue), SrcAddr:=ADR(uiValue), Write := TRUE );
	IF NOT Write_ADS.BUSY 
	THEN
		IF Write_ADS.ERR
		THEN
			MemError										:= TRUE;
			LastErrorState									:= state;
			LastErrorId										:= Read_Ads.ERRID;				
			State											:= 600; //Jump to state 600 to restore old entrys
		ELSE
			state											:= state + 1;
		END_IF
		Write_ADS(Write := FALSE);						
	END_IF
	
203:	
	uiValue													:= TO_UINT(FALSE);
	Write_ADS(NetId:= '' , Port:=500, IdxGrp:=16#5000+Axis.NcToPlc.AxisId, IDxOffs:=16#B,
					LEN:=SIZEOF(uiValue), SrcAddr:=ADR(uiValue), Write := TRUE );
	IF NOT Write_ADS.BUSY 
	THEN
		IF Write_ADS.ERR
		THEN
			MemError										:= TRUE;
			LastErrorState									:= state;
			LastErrorId										:= Read_Ads.ERRID;				
			State											:= 600; //Jump to state 600 to restore old entrys
		ELSE
			state											:= 204;
		END_IF
		Write_ADS(Write := FALSE);						
	END_IF

	
204://Write the max torque value used for homing
	IF DrvChannel = 1
	THEN
		CoERead.Index										:= SEL(DriveProfileIsDS402, 16#7110 , 	16#6872); 
		CoERead.SubIndex									:= SEL(DriveProfileIsDS402, 16#B  , 	16#0);
	ELSE //Channel 0
		CoERead.Index										:= SEL(DriveProfileIsDS402, 16#7010 , 	16#6072);
		CoERead.SubIndex									:= SEL(DriveProfileIsDS402, 16#B  , 	16#0);
 	END_IF 

	uiValue													:= LREAL_TO_UINT(MaxTorque) * 10;
	CoEWrite(
		NetId			:= '', 
		Index			:= , //See above
		SubIndex		:= , //See above
		pSrcBuf			:= ADR(uiValue), 
		BufLen			:= SIZEOF(uiValue),//2, 
		Execute			:= TRUE, 
		Axis			:= Axis
	);
	IF NOT CoEWrite.BUSY 
	THEN
		IF CoEWrite.Error
		THEN
			MemError										:= TRUE;
			LastErrorState									:= state;
			LastErrorId										:= CoEWrite.AdsErrId;//or CANopenErrId;				
			State											:= 600; //Jump to state 600 to restore old entrys
		ELSE
			state											:= 300;
		END_IF
		CoEWrite(Execute := FALSE, Axis := Axis);						
	END_IF
	
(* Velocity move until Homing_Tolerance exceeded *****************************************************************)
300:
	MC_Velocity( 
		Axis			:= Axis,
		Execute			:= TRUE,
		Velocity		:= VelocityTowardsBlock,
		Direction		:= Direction,
		Acceleration	:= Acceleration,
		Deceleration	:= Deceleration
	);
	
	IF ABS(Axis.NcToPlc.PosDiff) > lagTolerance
		OR NOT MC_Velocity.Busy //In case and error occure, the state machine can still continie
	THEN
		IF MC_Velocity.Error
		THEN
			MemError										:= TRUE;
			LastErrorState									:= state;
			LastErrorId										:= MC_Velocity.ErrorID;	
			state											:= 600; //Try to restore old parameter first
		ELSE
			MemBlockPos										:= Axis.NcToPlc.ActPos; //Record block pos
			MC_Halt(Execute := TRUE, Axis := Axis);
			State 											:= state + 1;
		END_IF
		MC_Velocity(Execute := FALSE, Axis := Axis);
	END_IF
	
301: //Wait for movment stopped 
	MC_Halt(Execute := TRUE, Axis := Axis);
	IF NOT MC_Halt.Busy
	THEN
		IF MC_Halt.Error
		THEN
			MemError										:= TRUE;
			LastErrorState									:= state;
			LastErrorId										:= MC_Halt.ErrorID;	
			state											:= 600; //Try to restore old parameter first		
		ELSE	
			state											:= 400; 	
		END_IF
		MC_Halt(Execute := FALSE, Axis := Axis);
	END_IF
	
400://Move to offset 
	MC_Absolute(
		Axis			:= Axis,
		Execute			:= TRUE,		
		Position		:= MemBlockPos + (ABS(Offset) * SEL(MC_Velocity.Direction = MC_Negative_Direction, -1.0 , 1.0)), //Calculate offset direction automaically 
		Velocity		:= VelocityOffBlock,
		Acceleration	:= Acceleration,
		Deceleration	:= Deceleration
	);
	IF NOT MC_Absolute.Busy 
	THEN
		IF MC_Absolute.Error
		THEN
			MemError										:= TRUE;
			LastErrorState									:= state;
			LastErrorId										:= MC_Absolute.ErrorID;	
			state											:= 600; //Try to restore old parameter first		
		ELSE	
			state											:= 500; 	
		END_IF
		MC_Absolute(Execute := FALSE, Axis := Axis);
	END_IF
	
500://Set home position and home flag
	IF Position <> DEFAULT_HOME_POSITION
	THEN
		MC_Home.Position									:= Position + (ABS(MemBlockPos - Axis.NcToPlc.ActPos) * SEL(MC_Velocity.Direction = MC_Negative_Direction, -1.0 , 1.0));
	ELSE
		MC_Home.Position									:= Param_CalibrationValue + (ABS(MemBlockPos - Axis.NcToPlc.ActPos) * SEL(MC_Velocity.Direction = MC_Negative_Direction, -1.0 , 1.0)); 
	END_IF
	MC_Home(
		Axis 		:= Axis,
		Execute		:= TRUE,
		Position	:= , //see above 
		HomingMode	:= MC_Direct
	);
	IF NOT MC_Home.Busy 
	THEN
		IF NOT MC_Home.Error
		THEN
			MemError										:= TRUE;
			LastErrorState									:= state;
			LastErrorId										:= MC_Absolute.ErrorID;	
			state											:= 600; //Try to restore old parameter first			
		ELSE
			state											:= 600;
		END_IF
		MC_Home(Execute := FALSE, Axis := Axis);
	END_IF

(* Return parameters for NC and drive to prior value ************************************************)
600:
	uiValue													:= TO_UINT(Param_MotionMonitoring.1);
	Write_ADS(NetId:= '' , Port:=500, IdxGrp:=16#4000+Axis.NcToPlc.AxisId, IDxOffs:=16#11,
				LEN:=SIZEOF(uiValue), SrcAddr:=ADR(uiValue), Write := Param_MotionMonitoring.0 );
	IF NOT Write_ADS.BUSY 
	THEN
		IF Write_ADS.ERR AND NOT MemError
		THEN
			MemError										:= TRUE;
			LastErrorState									:= state;
			LastErrorId										:= Write_ADS.ERRID;	
		END_IF
		Write_ADS(Write := FALSE);
		State												:= state + 1;									
	END_IF
		
601:
	uiValue													:= TO_UINT(Param_LagMonitoring.1);	
	Write_ADS(NetId:= '' , Port:=500, IdxGrp:=16#6000+Axis.NcToPlc.AxisId, IDxOffs:=16#10,
				LEN:=SIZEOF(uiValue), SrcAddr:=ADR(uiValue), Write := Param_LagMonitoring.0 );
	IF NOT Write_ADS.BUSY 
	THEN
		IF Write_ADS.ERR AND NOT MemError
		THEN
			MemError										:= TRUE;
			LastErrorState									:= state;
			LastErrorId										:= Write_ADS.ERRID;	
		END_IF
		Write_ADS(Write := FALSE);
		State												:= state + 1;									
	END_IF
	
602:
	uiValue													:= TO_UINT(Param_SoftMaxMonitoring.1);
	Write_ADS(NetId:= '' , Port:=500, IdxGrp:=16#5000+Axis.NcToPlc.AxisId, IDxOffs:=16#C,
				LEN:=SIZEOF(uiValue), SrcAddr:=ADR(uiValue), Write := Param_SoftMaxMonitoring.0 );
	IF NOT Write_ADS.BUSY 
	THEN
		IF Write_ADS.ERR AND NOT MemError
		THEN
			MemError										:= TRUE;
			LastErrorState									:= state;
			LastErrorId										:= Write_ADS.ERRID;	
		END_IF
		Write_ADS(Write := FALSE);
		State												:= state + 1;									
	END_IF
	
603:
	uiValue													:= TO_UINT(Param_SoftMinMonitoring.1);
	Write_ADS(NetId:= '' , Port:=500, IdxGrp:=16#5000+Axis.NcToPlc.AxisId, IDxOffs:=16#B,
				LEN:=SIZEOF(uiValue), SrcAddr:=ADR(uiValue), Write := Param_SoftMinMonitoring.0 );
	IF NOT Write_ADS.BUSY 
	THEN
		IF Write_ADS.ERR AND NOT MemError
		THEN
			MemError										:= TRUE;
			LastErrorState									:= state;
			LastErrorId										:= Write_ADS.ERRID;	
		END_IF
		Write_ADS(Write := FALSE);
		State												:= 604;									
	END_IF

604:
	IF DrvChannel = 1
	THEN
		CoERead.Index										:= SEL(DriveProfileIsDS402, 16#7110 , 	16#6872); 
		CoERead.SubIndex									:= SEL(DriveProfileIsDS402, 16#B  , 	16#0);
	ELSE //Channel 0
		CoERead.Index										:= SEL(DriveProfileIsDS402, 16#7010 , 	16#6072);
		CoERead.SubIndex									:= SEL(DriveProfileIsDS402, 16#B  , 	16#0);
 	END_IF 

	uiValue													:= Param_MaxTorque;
	CoEWrite(
		NetId			:= '', 
		Index			:= ,//See above
		SubIndex		:= , //See above 
		pSrcBuf			:= ADR(uiValue), 
		BufLen			:= SIZEOF(uiValue),//2,
		Execute			:= Param_MaxTorqueRead, 
		Axis			:= Axis
	);
	IF NOT CoEWrite.BUSY 
	THEN
		IF CoEWrite.Error
		THEN
			MemError										:= TRUE;
			LastErrorState									:= state;
			LastErrorId										:= CoEWrite.AdsErrId;//or CANopenErrId;				
		END_IF
		CoEWrite(Execute := FALSE, Axis := Axis);
		state												:= 900;			
	END_IF
	
(* Done *****************************************************************************)
900://Wait for execute signal to change to false
	Done 													:= NOT MemError; //Set the done flag to true if not error occur
	BUSY 													:= FALSE;
	Error													:= MemError;
	ErrorId													:= SEL(Error, 0 , LastErrorId);
	
	//Make sure all components stop operating
	Read_ADS(Read := FALSE);	Write_Ads(Write := FALSE);
	CoEWrite(Execute := FALSE,axis  := axis); CoERead(Execute := FALSE,axis  := axis);	
	MC_Home(Execute := FALSE,Axis := Axis);
	MC_Halt(Execute := FALSE,Axis := Axis);
	MC_Velocity(Execute := FALSE,Axis := Axis);
	MC_Absolute(Execute := FALSE,Axis := Axis);	
	
	State													:= 0;
END_CASE

END_FUNCTION_BLOCK

// ---- POUs/Motion/TF50xx-NC/02_Options/Phasing/AxPhasing.TcPOU
{attribute 'no_check'}
//Nc-axis phasing control 
//based on Tc2_MC2 library
FUNCTION_BLOCK AxPhasing EXTENDS AxFbBase
VAR_OUTPUT CONSTANT
	FNC_HALT_PHASING										:	INT := 0;
	FNC_PHASING_ABSOULTE									:	INT := 1;
	FNC_PHASING_RELATIVE									:	INT := 2;
END_VAR               
VAR_INPUT								
	Fnc														:	INT (FNC_HALT_PHASING..FNC_PHASING_RELATIVE) := FNC_HALT_PHASING;
	PhaseShift												:	LREAL := 0;
	Velo													:	LREAL := 0;
	Acc														:	LREAL := 0.0; // if Acc = 0, the NC-Value will be set                        								
	Dec														:	LREAL := 0.0; // if Dec = 0, the NC-Value will be set
	Jerk													:	LREAL := 0.0; // if Jerk = 0, the NC-Value will be set
	BufferMode												:	MC_BufferMode := MC_Aborting;(* 	MC_Aborting,
																									MC_Buffered,
																									MC_BlendingLow,
																									MC_BlendingPrevious,
																									MC_BlendingNext,
																									MC_BlendingHigh *)
                            								                        								
	Options 												: 	ST_PhasingOptions;
	rMasterAxis												:	REFERENCE TO AXIS_REF := 0;
END_VAR                     								
VAR_IN_OUT                  								
END_VAR                     									
VAR_OUTPUT                  	
	AbsolutePhaseShift										:	LREAL;
	CoveredPhaseShift										:	LREAL;
END_VAR
VAR
(* Zwischenspeicher **************************************************************************)
	MemFnc													:	INT := -1;

(* Trigger *)

(* Instanzierung der MC Bausteine *******************************************************)
	MC_HaltPhasing											:	MC_HaltPhasing;
	MC_PhasingAbsolute										:	MC_PhasingAbsolute;
	MC_PhasingRelative										:	MC_PhasingRelative;

(* Dummy Speicher **********************************************************)
(*	i,j		: INT := 0 ; *)
END_VAR

	(************************************************************************************)
	(*																					*)
	(*		B E C K H O F F   N E W   A U T O M A T I O N   T E C H N O L O G Y    		*)
	(*																					*)
	(*		Eiserstr.5	D-33415 Verl	Germany	phone:	+49-5246-0	www.Beckhoff.Com	*)
    (*																					*)
    (*		Bausteinbeschreibung	:	Gear axis function-block						*)
	(*		TwinCAT-Version			:	3.x or higher		 							*)
	(*		Version					:	V1.0 / 04/16									*)
 	(*		Autor					:	Thorsten Hemel									*)
	(*																					*)
	(************************************************************************************)

(* Execute ***************************************************************************************)
	rtExecute(CLK := Execute);
	IF rtExecute.Q
		AND MemFnc < 0
	THEN
		MemFnc 												:= Fnc ;
		Busy												:= TRUE;
		Done												:= FALSE;
		Active												:= FALSE;
		Error												:= FALSE;
		ErrorID												:= 0;
		CmdAborted											:= FALSE;
		ErrorText											:= '';
	END_IF

(* Call Method ***********************************************************************************)
	CASE MemFnc OF
	FNC_HALT_PHASING:
		HaltPhasing(Execute);

	FNC_PHASING_ABSOULTE:
		PhasingAbsoulte(Execute);

	FNC_PHASING_RELATIVE:
		PhasingRelative(Execute);

	-1:
		IF NOT Execute
		THEN
			Busy											:= FALSE;
			Done											:= FALSE;
			Active											:= FALSE;
			Error											:= FALSE;
			ErrorID											:= 0;
			CmdAborted										:= FALSE;
			ErrorText										:= '';
		END_IF                              				
	ELSE                                    				
		Busy												:= FALSE;
		Done												:= FALSE;
		Active												:= FALSE;
		Error												:= Execute;
		ErrorID												:= E_AdsErr.DEVICE_INVALIDPARM;
		CmdAborted											:= FALSE;
		ErrorText											:= CONCAT('invalid parameter value(s) Fnc no: ' , INT_TO_STRING(MemFnc));
	END_CASE                            		
                                            	

(*************************************************************************************************)

METHOD PUBLIC haltPhasing : BOOL //Return value = TRUE if busy
//required parameter
//rAxis
//rMasterAxis1
//RatioNumerator
//RatioDenominator
//Acc
//Dec
//Jerk
VAR_INPUT
	Execute													:	BOOL;
END_VAR
MemFnc 														:= FNC_HALT_PHASING;
THIS^.Execute												:= Execute;

IF NOT __ISVALIDREF(rAxis) 
THEN
	Busy													:= NOT Error;
	Error													:= TRUE;
	ErrorId													:= E_AdsErr.DEVICE_INVALIDPARM;
	CmdAborted												:= FALSE;
	Done													:= FALSE;
	Active													:= FALSE;
	ErrorText												:= 'Reference rAxis invalid (0)';
	MemFnc													:= SEL(Execute , -1 ,MemFnc); 
	RETURN;
ELSIF NOT __ISVALIDREF(rMasterAxis)
THEN
	Busy													:= NOT Error;
	Error													:= TRUE;
	ErrorId													:= E_AdsErr.DEVICE_INVALIDPARM;
	CmdAborted												:= FALSE;
	Done													:= FALSE;
	ErrorText												:= 'Reference rMasterAxis invalid (0)';
	MemFnc													:= SEL(Execute , -1 ,MemFnc); 
	RETURN;
END_IF

	MC_HaltPhasing(
		Execute				:= Execute, 
		Master				:= rMasterAxis, 
		Slave				:= rAxis, 
		Deceleration		:= Dec, 
		Jerk				:= Jerk, 
		BufferMode			:= BufferMode, 
		Options				:= Options, 
		Done				=> Done, 
		Busy				=> Busy, 
		Active				=> Active, 
		CommandAborted		=> CmdAborted, 
		Error				=> Error, 
		ErrorID				=> ErrorID);

	IF Error THEN
		LastErrorId											:= ErrorID;
		ErrorText 											:= CONCAT('Error MC_HaltPhasing ID:' , UDINT_TO_STRING(ErrorId));
	ELSE
		ErrorText 											:= '';
	END_IF

	IF NOT Execute AND NOT Busy
	THEN
		MemFnc												:=  -1;
	END_IF
	
	haltPhasing												:= Busy;
END_METHOD

METHOD PUBLIC phasingAbsoulte : BOOL //Return value = TRUE if busy
//required parameter
//rAxis
//rMasterAxis
//PhaseShift
//Acc
VAR_INPUT
	Execute													:	BOOL;
END_VAR
MemFnc 														:= FNC_PHASING_ABSOULTE;
THIS^.Execute												:= Execute;

IF NOT __ISVALIDREF(rAxis) 
THEN
	Busy													:= NOT Error;
	Error													:= TRUE;
	ErrorId													:= E_AdsErr.DEVICE_INVALIDPARM;
	CmdAborted												:= FALSE;
	Done													:= FALSE;
	Active													:= FALSE;
	ErrorText												:= 'Reference rAxis invalid (0)';
	MemFnc													:= SEL(Execute , -1 ,MemFnc); 
	RETURN;
ELSIF NOT __ISVALIDREF(rMasterAxis)
THEN
	Busy													:= NOT Error;
	Error													:= TRUE;
	ErrorId													:= E_AdsErr.DEVICE_INVALIDPARM;
	CmdAborted												:= FALSE;
	Done													:= FALSE;
	ErrorText												:= 'Reference rMasterAxis1 invalid (0)';
	MemFnc													:= SEL(Execute , -1 ,MemFnc); 
	RETURN;
END_IF

	MC_PhasingAbsolute(
		Execute				:= Execute, 
		Master				:= rMasterAxis, 
		Slave				:= rAxis, 
		PhaseShift			:= PhaseShift, 
		Velocity			:= Velo, 
		Acceleration		:= Acc, 
		Deceleration		:= Dec, 
		Jerk				:= Jerk, 
		BufferMode			:= BufferMode, 
		Options				:= Options, 
		Done				=> Done, 
		Busy				=> Busy, 
		Active				=> Active, 
		CommandAborted		=> CmdAborted, 
		Error				=> Error, 
		ErrorID				=> ErrorId, 
		AbsolutePhaseShift	=> AbsolutePhaseShift);
		

	IF Error THEN
		LastErrorId											:= ErrorID;
		ErrorText 											:= CONCAT('Error MC_PhasingAbsolute ID:' , UDINT_TO_STRING(ErrorId));
	ELSE
		ErrorText 											:= '';
	END_IF

	IF NOT Execute AND NOT Busy
	THEN
		MemFnc												:=  -1;
	END_IF
	
	phasingAbsoulte											:= Busy;
END_METHOD

METHOD PUBLIC phasingRelative : BOOL//Return value = TRUE if busy
//required parameter
//rAxis
//rMasterAxis
//PhaseShift
//Acc
VAR_INPUT
	Execute													:	BOOL;
END_VAR
MemFnc														:= FNC_PHASING_RELATIVE;
THIS^.Execute												:= Execute;
	                										
IF NOT __ISVALIDREF(rAxis) 
THEN
	Busy													:= NOT Error;
	Error													:= TRUE;
	ErrorId													:= E_AdsErr.DEVICE_INVALIDPARM;
	CmdAborted												:= FALSE;
	Done													:= FALSE;
	Active													:= FALSE;
	ErrorText												:= 'Reference rAxis invalid (0)';
	MemFnc													:= SEL(Execute , -1 ,MemFnc); 
	RETURN;
ELSIF NOT __ISVALIDREF(rMasterAxis)
THEN
	Busy													:= NOT Error;
	Error													:= TRUE;
	ErrorId													:= E_AdsErr.DEVICE_INVALIDPARM;
	CmdAborted												:= FALSE;
	Done													:= FALSE;
	ErrorText												:= 'Reference rMasterAxis invalid (0)';
	MemFnc													:= SEL(Execute , -1 ,MemFnc); 
	RETURN;	
END_IF
	

	MC_PhasingRelative( 
		Execute				:= Execute,
		Master				:= rMasterAxis, 
		Slave				:= rAxis, 
		PhaseShift			:= PhaseShift, 
		Velocity			:= Velo, 
		Acceleration		:= Acc, 
		Deceleration		:= Dec, 
		Jerk				:= Jerk, 
		BufferMode			:= BufferMode, 
		Options				:= Options, 
		Done				=> Done, 
		Busy				=> Busy, 
		Active				=> Active, 
		CommandAborted		=> CmdAborted, 
		Error				=> Error, 
		ErrorID				=> ErrorId, 
		CoveredPhaseShift	=> CoveredPhaseShift);					

	IF Error THEN
		LastErrorId											:= ErrorID;
		ErrorText 											:= CONCAT('Error MC_PhasingRelative ID:' , UDINT_TO_STRING(ErrorId));
	ELSE
		ErrorText 											:= '';
	END_IF

	IF NOT Execute AND NOT Busy
	THEN
		MemFnc												:=  -1;
	END_IF
	
	phasingRelative												:= Busy;
END_METHOD

END_FUNCTION_BLOCK

// ---- POUs/Motion/TF50xx-NC/02_Options/TouchProbe/AxTouchProbe.TcPOU
{attribute 'no_check'}
//Nc-axis touch probe  
//based on Tc2_MC2 library
FUNCTION_BLOCK AxTouchProbe EXTENDS AxFbBase
VAR_OUTPUT CONSTANT
	FNC_RUN													:	INT := 0;
	FNC_ABORT												:	INT := 1;
END_VAR                     								
VAR_INPUT                   								
	Fnc														: 	INT (FNC_RUN..FNC_ABORT):= FNC_RUN;
	TriggerInput											: 	TRIGGER_REF;
	WindowOnly												: 	BOOL := FALSE;(* Enables the monitoring window *)
	FirstPosition											: 	LREAL;	(* Beginning of the monitoring window *)
	LastPosition 											: 	LREAL;	(* Ending of the monitoring window *)
END_VAR
VAR_IN_OUT
END_VAR
VAR_OUTPUT
	RecordedPosition										: 	LREAL;	// current axisposition on trigger-event
	RecordedData											:	MC_TouchProbeRecordedData;
END_VAR
VAR
(* cache **************************************************************************)
	MemFnc													:	INT := -1;
               								                           	
(* trigger *)               	

(* MC-function-block instances ****************************************************)
	MC_TouchProbe											: 	MC_TouchProbe;
	MC_AbortTrigger											:	MC_AbortTrigger;

END_VAR

	(************************************************************************************)
	(*																					*)
	(*		B E C K H O F F   N E W   A U T O M A T I O N   T E C H N O L O G Y    		*)
	(*																					*)
	(*		Eiserstr.5	D-33415 Verl	Germany	phone:	+49-5246-0	www.Beckhoff.Com	*)
    (*																					*)
    (*		Bausteinbeschreibung	:	TouchProbe ctrl									*)
	(*		TwinCAT-Version			:	3.x or higher 									*)
	(*		Version					:	V3.0 / 03/13									*)
	(*		Lib						:	TcMC2.lib 										*)
 	(*		Autor					:	DSC												*)
	(*																					*)
	(************************************************************************************)

(* Execute ***************************************************************************************)
	rtExecute(CLK := Execute);
	IF rtExecute.Q
		AND MemFnc < 0
	THEN
		MemFnc 												:= SEL(Fnc = FNC_RUN, FNC_ABORT , FNC_RUN) ;
		Busy												:= TRUE;
		Done												:= FALSE;
		Error												:= FALSE;
		ErrorID												:= 0;
		CmdAborted											:= FALSE;
	END_IF

(* Call Method ***********************************************************************************)
	CASE MemFnc OF
	FNC_RUN:
		Run(Execute);

	FNC_ABORT:
		Abort(Execute);

	-1:
		IF NOT Execute
		THEN
			Busy											:= FALSE;
			Done											:= FALSE;
			Error											:= FALSE;
			ErrorID											:= 0;
			CmdAborted										:= FALSE;
		END_IF                              				
	ELSE                                    				
		Busy												:= FALSE;
		Done												:= FALSE;
		Error												:= Execute;
		ErrorID												:= E_AdsErr.DEVICE_INVALIDPARM;
		CmdAborted											:= FALSE;
	END_CASE                                	

(*************************************************************************************************)

METHOD PUBLIC abort : BOOL //Return value = TRUE if busy
//required parameter
//rAxis
//TriggerInput
VAR_INPUT
	Execute													:	BOOL := FALSE;
END_VAR
	MemFnc	 												:= FNC_ABORT;
	THIS^.Execute											:= Execute;
IF NOT __ISVALIDREF(rAxis) 
THEN
	Busy													:= NOT Error;
	ErrorId													:= E_AdsErr.DEVICE_INVALIDPARM;
	Error													:= TRUE;
	Done													:= FALSE;
	CmdAborted												:= FALSE;
	MemFnc													:= SEL(Execute , -1 ,MemFnc); 
	RETURN;
END_IF

	MC_AbortTrigger(
		Execute		:= Execute,
		Axis		:= rAxis,
		TriggerInput:= TriggerInput,
		Done		=> done,
		Busy		=> Busy,
		Error		=> Error,
		ErrorID		=> ErrorID);

	CmdAborted		:= FALSE;

	IF NOT Execute AND NOT Busy
	THEN
		MemFnc												:= -1;
	END_IF                              					
	                                    	
	abort 													:= Busy;
END_METHOD

METHOD PUBLIC run : BOOL //Return value = TRUE if busy
//required parameter
//rAxis
//TriggerInput
//WindowOnly
//FirstPosition
//LastPosition
VAR_INPUT
	Execute													: BOOL := FALSE;
END_VAR
	MemFnc 													:= FNC_RUN;
	THIS^.Execute											:= Execute;
	
IF NOT __ISVALIDREF(rAxis) 
THEN
	Busy													:= NOT Error;
	ErrorId													:= E_AdsErr.DEVICE_INVALIDPARM;
	Error													:= TRUE;
	Done													:= FALSE;
	CmdAborted												:= FALSE;
	MemFnc													:= SEL(Execute , -1 ,MemFnc); 
	RETURN;
END_IF

	MC_TouchProbe(
		Execute			:= Execute,
		WindowOnly		:= WindowOnly,
		FirstPosition	:= FirstPosition,
		LastPosition	:= LastPosition,
		Axis			:= rAxis,
		TriggerInput	:= TriggerInput,
		Done			=> Done,
		Busy			=> Busy,
		CommandAborted	=> CmdAborted,
		Error			=> Error,
		ErrorID			=> ErrorID,
		RecordedPosition=> RecordedPosition,
		RecordedData 	=> RecordedData);

	IF NOT Execute AND NOT Busy
	THEN
		MemFnc												:= -1;
	END_IF
	
	run														:= busy;
END_METHOD

END_FUNCTION_BLOCK

// ---- POUs/Motion/TF50xx-NC/03_Utilities/AxAutoFct.TcPOU
{attribute 'no_check'}
FUNCTION_BLOCK AxAutoFct
VAR_INPUT
	Enable													:	BOOL := FALSE;(* Enable block *)
	AutoInit												:	BOOL := TRUE; (* TRUE=With Enable force status will be written to axis / FALSE=Force values will only be written on change *) 
	AxisId													: 	DWORD; (* ID der Achse *)
	ForceSoftLimit											:	BOOL := TRUE; (* TRUE => SoftLimitMonitoring = True *)
	ForceCalibration										:	BOOL := FALSE;(* TRUE => Calibrated = True  *)
	ForcePosLagMon											:	BOOL := TRUE; (* TRUE => Position Lag Monitoring = True  *)
	ForcePosMon												:	BOOL := TRUE; (* TRUE => In Position Monitoring = True  *)
	ForceTargetMon											:	BOOL := TRUE; (* TRUE => In Target Monitoring = True  *)
END_VAR                         							
VAR_IN_OUT                      							
END_VAR                         							
VAR_OUTPUT        
	{attribute 'displaymode':='binary'}              							
	Status													:	BYTE := 0;
	Busy													:	BOOL := FALSE;
	Error													:	BOOL := FALSE;
	ErrorID													:	UDINT := 0;
END_VAR                         	

VAR
(* Cache **********************************************************************)
	State													: 	INT;
	InitDone												:	BYTE;
	LastErrText												:	STRING(20);
	
(* Instances *******************************************************************)
	WriteAdsPara											: 	ADSWRITE := (NetID:= '' , Port:=AMSPORT_R0_NC, TmOut	:= DEFAULT_ADS_TIMEOUT);

(* Dummy  *********************************************************************)
	tmpWORD													:	UINT;

END_VAR

	(* Enable/Disable of: Soft limit monitoring, Target monitoring, Pos. Lag monitoring,  Calibration 	*)
	(*																									*)
	(****************************************************************************************************)

(* writing parameters *******************************************************************************)
IF NOT Enable 
THEN
	Status.0 												:= NOT forceSoftLimit;
	Status.1 												:= NOT forceCalibration;
	Status.2 												:= NOT forcePosLagMon;
	Status.3 												:= NOT forcePosMon;
	Status.4 												:= NOT forceTargetMon;
	            											
	InitDone 												:= SEL(AutoInit , 2#0001_1111 , 2#0000_0000);
                											
	State 													:= 0;
	Error													:= FALSE;
	ErrorID													:= 0;
	Busy 													:= FALSE;
ELSIF AxisId = 0 
THEN
	ErrorID													:= E_AdsErr.DEVICE_INVALIDPARM;
	Error													:= FALSE;
	Busy													:= FALSE;
ELSE
	CASE State OF
	0:	(* Init *)

		Busy := FALSE;

		IF NOT WriteAdsPara.BUSY
			AND NOT WriteAdsPara.WRITE
		 	AND NOT Error
		THEN
			IF (forceSoftLimit XOR status.0) OR NOT InitDone.0 THEN
				InitDone.0 									:= TRUE;
				status.0 									:= forceSoftLimit;
				tmpWord 									:= BOOL_TO_UINT(forceSoftLimit);
				State 										:= 1;
				Busy 										:= TRUE;

			ELSIF(forceCalibration XOR status.1) OR NOT InitDone.1 THEN
				InitDone.1 									:= TRUE;
				status.1 									:= forceCalibration;
				tmpWord 									:= BOOL_TO_UINT(forceCalibration);
				State 										:= 10;
				Busy 										:= TRUE;
	
			ELSIF(forcePosLagMon XOR status.2) OR NOT InitDone.2 THEN
				InitDone.2 									:= TRUE;
				status.2 									:= forcePosLagMon;
				tmpWord 									:= BOOL_TO_UINT(forcePosLagMon);
				State 										:= 20;
				Busy 										:= TRUE;
			ELSIF(forcePosMon XOR status.3) OR NOT InitDone.3 THEN
				InitDone.3 									:= TRUE;
				status.3 									:= forcePosMon;
				tmpWord 									:= BOOL_TO_UINT(forcePosMon);
				State 										:= 30;
				Busy 										:= TRUE;
			ELSIF(forceTargetMon XOR status.4) OR NOT InitDone.4 THEN
				InitDone.4 									:= TRUE;
				status.4 									:= forceTargetMon;
				tmpWord 									:= BOOL_TO_UINT(forceTargetMon);
				State 										:= 40;
				Busy 										:= TRUE;
		
			END_IF
		ELSE
			WriteAdsPara	(Write := FALSE);
		END_IF

	1: (* toggle positive limit switches ****************************************************************)
		IF NOT WriteAdsPara.Busy
			AND WriteAdsPara.Write
		THEN
			IF WriteAdsPara.Err THEN
				State 										:= 9999;  // goto Error-state 
			ELSE           									
				State 										:= State + 1;
			END_IF         	
		END_IF

		WriteAdsPara(
			IdxGrp	:=16#4000+AxisId,
			IdxOffs	:=16#1000C,
			LEN		:=SIZEOF(tmpWord),
			SrcAddr	:=ADR(tmpWord),
			Write 	:= State = 1);

	2: (* toggle negative limit switches *****************************************************************)
		IF NOT WriteAdsPara.Busy
			AND WriteAdsPara.Write
		THEN
			IF WriteAdsPara.Err THEN
				State 										:= 9999; // goto Error-state 
			ELSE
				State 										:= 99; // done 
			END_IF
		END_IF

		WriteAdsPara(
			IdxGrp	:=16#4000+AxisId,
			IdxOffs	:=16#1000B,
			LEN		:=SIZEOF(tmpWord),
			SrcAddr	:=ADR(tmpWord),
			Write 	:= State = 2);

	10: (* set referenceflag *****************************************************************)
		IF NOT WriteAdsPara.Busy
			AND WriteAdsPara.Write
		THEN
			IF WriteAdsPara.Err THEN
				State 										:= 9999;  	// goto Error-state 
			ELSE           									
				State 										:= 99; 		// done 
			END_IF
		END_IF

		WriteAdsPara(
			IdxGrp	:=16#5100+AxisId,
			IdxOffs	:=16#9,
			LEN		:=SIZEOF(tmpWord),
			SrcAddr	:=ADR(tmpWord),
			Write 	:= State = 10 );
			
	20: (* lagdistance monitoring *****************************************************************)
		IF NOT WriteAdsPara.Busy
			AND WriteAdsPara.Write
		THEN
			IF WriteAdsPara.Err THEN
				State 										:= 9999;  	// goto Error-state 
			ELSE           									
				State 										:= 99; 		// done
			END_IF
		END_IF

		WriteAdsPara(
			IdxGrp	:=16#6000+AxisId,
			IdxOffs	:=16#10,
			LEN		:=SIZEOF(tmpWord),
			SrcAddr	:=ADR(tmpWord),
			Write 	:= State = 20);
			
	30: (* Position Monitoring *****************************************************************)
		IF NOT WriteAdsPara.Busy
			AND WriteAdsPara.Write
		THEN
			IF WriteAdsPara.Err THEN
				State 										:= 9999;  	// goto Error-state 
			ELSE           									
				State 										:= 99; 		// done
			END_IF
		END_IF

		WriteAdsPara(

			IdxGrp	:=16#4000+AxisId,
			IdxOffs	:=16#F,
			LEN		:=SIZEOF(tmpWord),
			SrcAddr	:=ADR(tmpWord),
			Write 	:= State = 30 );

	40: (* Target Monitoring *****************************************************************)
		IF NOT WriteAdsPara.Busy
			AND WriteAdsPara.Write
		THEN
			IF WriteAdsPara.Err THEN
				State 										:= 9999;  	// goto Error-state 
			ELSE           									
				State 										:= 99; 		// done
			END_IF
		END_IF

		WriteAdsPara(
			IdxGrp	:=16#4000+AxisId,
			IdxOffs	:=16#15,
			LEN		:=SIZEOF(tmpWord),
			SrcAddr	:=ADR(tmpWord),
			Write 	:= State = 40 );
			
	ELSE (* case else *)
		IF WriteAdsPara.ERR THEN
			Error											:= TRUE;
			ErrorID											:= WriteAdsPara.ERRID;
			LastErrText										:= CONCAT('Err WriteAdsPara ID: ', UDINT_TO_STRING(ErrorID));
		ELSE            									
			State 											:= 0;
		END_IF
	END_CASE
END_IF

(************************************************************************************************************************)

END_FUNCTION_BLOCK

// ---- POUs/Motion/TF50xx-NC/03_Utilities/getOvrVelo.TcPOU
{attribute 'no_check'}
//Overwrite function - Returns velocity setpoint based on max velo and requested overwrite 
FUNCTION getOvrVelo : LREAL
VAR_INPUT
	SetVelo													:	LREAL;
	MaxVelo													:	LREAL;
END_VAR
VAR
END_VAR

IF 	MaxVelo = 0.0 OR SetVelo = 0.0
THEN
	GetOvrVelo 												:= 0.0;
ELSE                										
	GetOvrVelo 												:= 100.0 / MaxVelo * SetVelo;
END_IF

END_FUNCTION

// ---- POUs/Motion/TF50xx-NC/AxNcPTP.TcPOU
FUNCTION_BLOCK AxNcPTP EXTENDS AxNcBase implements I_AxNcPTP (* See Tc2_MC2 *)
VAR_OUTPUT CONSTANT
END_VAR
VAR_INPUT
	Motion													:	AxMotion;                                        
END_VAR                           
VAR_OUTPUT                  	
END_VAR
VAR

END_VAR

	(* Axis 																*)
	(************************************************************************)

	
(********************************************************************************)
(* Call AxNcBase																*)
(********************************************************************************)
	Super^();
		
(********************************************************************************)
(* work moving ctrl 															*)
(********************************************************************************)
	Motion(rAxis := THIS^);
	errorCheck(AxBase := Motion);
	
(********************************************************************************)

METHOD PUBLIC noAction : BOOL //Return value = TRUE if busy of home and motion 
VAR_INPUT
END_VAR

Motion.Execute	:= FALSE;
Motion.JogBwd	:= FALSE;
Motion.JogFwd	:= FALSE;

NoAction 		:= 	Super^.noAction() and NOT Motion.Busy;
END_METHOD

{attribute 'monitoring' := 'call'}
PROPERTY rMotion : REFERENCE TO AxMotion
GET
rMotion REF= Motion;
END_GET
END_PROPERTY

END_FUNCTION_BLOCK

// ---- POUs/StringHelper/DWORD_TO_BINSTR_EXT.TcPOU
{attribute 'no_check' := ''}
FUNCTION DWORD_TO_BINSTR_EXT : T_MaxString //This function converts a decimal number into a binary string (base 2), where the digits are separated according to the selected mode 
//e.g. 1111000011110000 -> 1111_0000_1111_0000 
VAR_INPUT
	In														: DWORD;//The decimal number requiring conversion.
	Precision												: INT; //Minimum number of displayed digits (digits), filled up with 0 from left if significant digits are less then that
	Mode													: INT; //1=Separate high and low word / 2=Separate bytes / 3=Separate nibbles /ELSE no separation | Separator = Param.DOWRD_TO_XXXSTR_EXT_SEPARATOR
END_VAR
VAR		
	k														:	INT;											
END_VAR

DWORD_TO_BINSTR_EXT 										:= DWORD_TO_BINSTR(in,precision);

CASE mode OF
1:// Separate by low word and high word
	DWORD_TO_BINSTR_EXT										:= INSERT_EXT(DWORD_TO_BINSTR_EXT, PARAM.XWORD_TO_XXXSTR_EXT_SEPARATOR ,16);
	
2://Separate by bytes
	DWORD_TO_BINSTR_EXT										:= INSERT_EXT(DWORD_TO_BINSTR_EXT,PARAM.XWORD_TO_XXXSTR_EXT_SEPARATOR,8);
	
3://Separate by nibble
	DWORD_TO_BINSTR_EXT										:= INSERT_EXT(DWORD_TO_BINSTR_EXT,PARAM.XWORD_TO_XXXSTR_EXT_SEPARATOR,4);
END_CASE

//Cut seperator at the end
k 															:= LEN(DWORD_TO_BINSTR_EXT);
IF k > 0 AND_THEN DWORD_TO_BINSTR_EXT[k-1] = PARAM.XWORD_TO_XXXSTR_EXT_SEPARATOR[0]
THEN
	DWORD_TO_BINSTR_EXT[k-1]								:= 0;
END_IF

END_FUNCTION

// ---- POUs/StringHelper/isWStringNumeric.TcPOU
{attribute 'no_check'}
//Returns TRUE in case a ascii string contains only a valid number signs. Minus,plus,space,comma and dot are allowed
//Limited to a Param.MAX_EXT_STRING_LENGTH long string  
FUNCTION isWStringNumeric : BOOL 
VAR_INPUT
	pSource													:	POINTER TO WORD;
END_VAR             										
VAR                 
	Cr														:	WORD;	//Char									
	countSeperator											:	INT;
	i														:	UDINT;
	Addr													:	POINTER TO WORD;
END_VAR

IF pSource <> 0
THEN
	isWStringNumeric										:=	TRUE;
	FOR i := 0 TO PARAM.MAX_EXT_STRING_LENGTH DO
		Addr												:= pSource + (i * 2);
		Cr												:= Addr^;
		IF Cr = 0
		THEN 														
			isWStringNumeric								:= i > 0; //Only TRUE if string is not empty 
			EXIT;
		ELSIF Cr = 46 OR Cr = 44 //comma or point as a seperator
		THEN
			countSeperator									:= countSeperator + 1;
			IF countSeperator > 1 
			THEN
				isWStringNumeric							:= FALSE;
				EXIT;	(* more than one seperator -> no number *)
			END_IF
		ELSIF(Cr < 48 OR Cr > 57)
			AND Cr <> 45 (* minus *)
			AND Cr <> 43 (* plus *)
			AND Cr <> 32 (* Space *)
			AND Cr <> 101(* e for 9.9999992e-2 *)
			OR i = PARAM.MAX_EXT_STRING_LENGTH
		THEN
			isWStringNumeric								:= FALSE;
			EXIT;	(* no numerical char *)
		END_IF
	END_FOR      
ELSE
	isWStringNumeric										:= FALSE;
END_IF

END_FUNCTION

// ---- POUs/StringHelper/replaceInString.TcPOU
{attribute 'no_check'}
//Replace a part of a string with another string 
FUNCTION replaceInString : BOOL
VAR_INPUT
	SearchStr												:	STRING(10); //e.g. '/r/n_
	ReplaceStr												:	STRING(10); //e.g. '-'
END_VAR             										
VAR_IN_OUT         										
	Strline													: 	T_MaxString;
END_VAR             										
VAR                 	
	StrLen, i,pos											:	INT;
END_VAR

IF strline = '' 
THEN 
	replaceInString											:= TRUE;
ELSE
	StrLen													:= LEN(strline);
	FOR i := 0 TO StrLen
	DO
		pos 												:= FIND(strline,SearchStr);
		IF pos >= 1 
		THEN
			strline											:= REPLACE(strline,ReplaceStr,LEN(SearchStr),pos);
		ELSE
			replaceInString									:= i > 0; 
			EXIT;						
		END_IF	
	END_FOR
END_IF

END_FUNCTION

// ---- POUs/StringHelper/ExtendedString/ExtWString.TcPOU
{attribute 'no_check' := ''}
FUNCTION_BLOCK ExtWString //WSTRING functions for a wstring with a lenght > 255. Lenght is defined by PARAM.MAX_EXT_STRING_LENGTH
VAR_OUTPUT CONSTANT
	MAX_LENGTH												: UDINT := PARAM.MAX_EXT_STRING_LENGTH;
END_VAR
VAR_OUTPUT
	ResultStr												: T_EXT_WSTRING;		
END_VAR
VAR
	str1Len													: UDINT;
 	str2Len													: UDINT; 
	cpyLenght												: UDINT;
END_VAR

//Concatenation (combination) of two extended wstrings (lenght definded by ET.Param.EXT_STRING_MAX_LENGHT)
METHOD CONCAT : UDINT //Returns the lenght of the new string
VAR_INPUT
	 rSTR1													:	REFERENCE TO T_EXT_WSTRING;
	 STR2													:	T_EXT_WSTRING;
	 rResult												:	REFERENCE TO T_EXT_WSTRING;
END_VAR
VAR_OUTPUT
END_VAR
VAR
END_VAR
MEMSET(ADR(ResultStr),0,SIZEOF(ResultStr));
IF __ISVALIDREF(rSTR1)
THEN
	str1Len 													:= LENGTH(rSTR1);
	str2Len 													:= LENGTH(STR2);
	MEMCPY(ADR(ResultStr), ADR(rSTR1), (str1Len + 1) * 2);	 //Copy first string to result
	cpyLenght													:= 1 + MIN(str2Len, MAX_LENGTH - str1Len);
	MEMCPY(ADR(ResultStr) + (2 * str1Len), ADR(STR2), SEL(cpyLenght >  1, 0, cpyLenght) * 2); //Add second string
	CONCAT														:= MIN(str1Len + str2Len,MAX_LENGTH);
	IF __ISVALIDREF(rResult) 
	THEN
		MEMCPY(ADR(rResult), ADR(ResultStr), 2 * (CONCAT + 1)); 
	END_IF
ELSE
	CONCAT														:= 0;
END_IF
END_METHOD

//The function DELETE removes a partial STRING from a larger WSTRING at a defined position. 
//The input variable rSTR is TYPE WSTRING with a lenght if ET.Param.EXT_STRING_MAX_LENGHT, LEN AND POS are TYPE UINT.
//The new string will be written into the result reference, in case of invalid pos or len parameter, the input string will be copied to rResult
//means: Delete LEN characters from rSTR beginning with the character in the POS
METHOD PUBLIC DELETE : UDINT //Returns the new string lenght
VAR_INPUT
	 rSTR													:	REFERENCE TO T_EXT_WSTRING;
	 LEN													:	UDINT (0..MAX_LENGTH) := 0;
	 POS													:	UDINT (0..MAX_LENGTH) := 0;
	 rResult												:	REFERENCE TO T_EXT_WSTRING;						
END_VAR
VAR
END_VAR
MEMSET(ADR(ResultStr),0,SIZEOF(ResultStr));
IF NOT __ISVALIDREF(rSTR) 
THEN
	DELETE													:= 0;
	RETURN;
END_IF

Str1Len 													:= THIS^.LENGTH(rSTR);
IF pos > 0 AND pos <= str1Len
THEN // Only executed if parameter within string limitation
	MEMCPY(ADR(ResultStr), ADR(rStr), MAX(0, POS -1 ) * 2); //First part of string
	cpyLenght 												:= Str1Len - MIN(Str1Len, MAX(0, POS -1 ) + LEN); 
	MEMCPY(ADR(ResultStr) + (2 * MAX(0,POS-1)), ADR(rStr) + (2 * MIN(Str1Len, POS -1 + LEN)), (cpyLenght + 1) * 2); //Second part of string
	DELETE													:= (cpyLenght - 1) + pos; //New string length
	IF __ISVALIDREF(rResult) 
	THEN
		MEMCPY(ADR(rResult), ADR(ResultStr), 2 * (DELETE + 1)); 
	END_IF
ELSE
	DELETE													:= Str1Len;
	IF __ISVALIDREF(rResult) 
	THEN
		MEMMOVE(ADR(rResult), ADR(rStr), 2 * (DELETE + 1)); 
	END_IF	
END_IF
END_METHOD

//FIND searches for a partial wstring within a wstring. FIND(STR1, STR2)
//means: Find the position of the first character where STR2 appears in STR1 for the first time. 
//If STR2 is not found in STR1, then FIND:=0.
METHOD PUBLIC FIND : UDINT //position of the first character where STR2 appears in STR1 for the first time.
VAR_INPUT
	 rSTR1													: REFERENCE TO T_EXT_WSTRING;
	 STR2													: T_EXT_WSTRING;
END_VAR
VAR
	 valid													: BOOL;
	 i, j													: UDINT;
END_VAR
FIND														:= 0;
IF NOT __ISVALIDREF(rSTR1) 
THEN
	RETURN;
END_IF

str1Len 													:= LENGTH(rSTR1);
str2Len 													:= LENGTH(STR2);
FOR i:= 0 TO str1Len 
DO
	IF rSTR1[i] = STR2[0] 
	THEN	// Wenn erstes Zeichen übereinstimmt
		valid												:= TRUE;
		FOR j := 1 TO str2Len - 1 DO // Alle zeichen von STR2 durchgehen
			valid 											:= rSTR1[i + j] = STR2[j];
			
			IF NOT valid THEN // Wenn Zeichen ungleich abbrechen
				RETURN;						
			END_IF	
		END_FOR
		FIND 												:= i + 1;
		RETURN;		
	END_IF
END_FOR
END_METHOD

//INSERT inserts a string into another wstring at a defined point.
//means: insert STR2 into STR1 after position POS.
METHOD PUBLIC INSERT : UDINT //Returns the lenght of the new string
VAR_INPUT
	 rSTR1													: REFERENCE TO T_EXT_WSTRING;
	 STR2													: T_EXT_WSTRING;
	 POS													: UDINT (0..MAX_LENGTH);  
	 rResult												: REFERENCE TO T_EXT_WSTRING;	
END_VAR
VAR
	 chkPos													: UDINT;	
END_VAR
MEMSET(ADR(ResultStr),0,SIZEOF(ResultStr));
IF NOT __ISVALIDREF(rSTR1) 
THEN
	INSERT													:= 0;
	RETURN;
END_IF
str1Len 													:= LENGTH(rSTR1);
str2Len 													:= LENGTH(STR2);
IF Pos >= 0 AND Pos <= Str1Len
THEN
	MEMCPY(ADR(ResultStr), ADR(rStr1), 2* (str1Len + 1));  //Copy string to to result
	chkPos 													:= LIMIT(0, POS, str1Len); //Limit insert pos to lenght string 1
	cpyLenght												:= MAX(0,MIN(str1Len - chkPos  + 1, MAX_LENGTH - chkPos - str2Len));
	MEMCPY(ADR(ResultStr) + (2 * (chkPos + str2Len)), ADR(rResult) + (2 * chkPos) ,2 * SEL(cpyLenght > 1, 0,cpyLenght)); //move rest of string 1 to the end
	cpyLenght												:= MIN(str2Len , MAX_LENGTH - chkPos);
	MEMCPY(ADR(ResultStr) + (2 * chkPos), ADR(Str2) ,cpyLenght * 2 );
	INSERT													:= MIN(MAX_LENGTH, str1Len + str2Len);
	IF __ISVALIDREF(rResult) 
	THEN
		MEMCPY(ADR(rResult), ADR(ResultStr), 2 * (INSERT + 1)); 
	END_IF
ELSE
	INSERT													:= str1Len;
	IF __ISVALIDREF(rResult) 
	THEN
		MEMMOVE(ADR(rResult), ADR(rStr1), 2 * (INSERT + 1)); 
	END_IF; 
END_IF
END_METHOD

//Left returns the left, initial wstring for a given string. LEFT (STR, SIZE) 
//means: Take the first SIZE character from the left in the string STR.
METHOD PUBLIC LEFT : UDINT
VAR_INPUT
	 rSTR													: REFERENCE TO T_EXT_WSTRING;
	 SIZE													: UDINT (0..MAX_LENGTH);
	 rResult												: REFERENCE TO T_EXT_WSTRING;
END_VAR
VAR_INPUT
	 
END_VAR
MEMSET(ADR(ResultStr),0,SIZEOF(ResultStr));
IF __ISVALIDREF(rSTR)
THEN
	SIZE													:= LIMIT(0,SIZE,MAX_LENGTH); 
	LEFT													:= MIN(LENGTH(rSTR), SIZE);
	MEMCPY(ADR(ResultStr), ADR(rSTR), 2 * LEFT);
	IF __ISVALIDREF(rResult) 
	THEN
		MEMCPY(ADR(rResult), ADR(ResultStr), 2 * (LEFT + 1)); 
	END_IF
ELSE
	LEFT													:= 0;
END_IF
END_METHOD

//Returns the length of a extended wstring.
METHOD PUBLIC LENGTH : UDINT
VAR_INPUT
	rSTR												:	REFERENCE TO T_EXT_WSTRING;
END_VAR
VAR
	i													:	UDINT;
END_VAR
IF __ISVALIDREF(rSTR) 
THEN
	LENGTH														:= 0;								
	FOR i := 0 TO MAX_LENGTH 
	DO
		IF rSTR[i] = 0 
		THEN
			LENGTH 											:= i;
			RETURN;
		END_IF
	END_FOR
ELSE
	LENGTH														:= 0;
END_IF
END_METHOD

//Mid returns a partial string from within a wstring. MID (STR, LEN, POS) 
//means: Retrieve LEN characters from the STR string beginning with the character at position POS.
METHOD PUBLIC MID : UDINT //Returns the lenght if the new string (result)
VAR_INPUT
	 rSTR													:	REFERENCE TO T_EXT_WSTRING;
	 LEN													:	UDINT (0..MAX_LENGTH) ;
	 POS													:	UDINT (0..MAX_LENGTH) ;
	 rResult												:	REFERENCE TO T_EXT_WSTRING;	
END_VAR
VAR
END_VAR
MEMSET(ADR(ResultStr),0,SIZEOF(ResultStr));
IF NOT __ISVALIDREF(rSTR)
THEN
	MID														:= 0;
	RETURN;	
END_IF

str1Len 													:= THIS^.LENGTH(rSTR);

IF POS >= 0 AND POS <= str1Len 
THEN	 
	cpyLenght 												:= MIN(str1Len - POS + 1, MIN(LEN, str1Len));	
	MEMMOVE(ADR(ResultStr), ADR(rSTR) + (2 * MAX(0,POS -1)), 2 * cpyLenght);
	MID														:=  cpyLenght;
	IF __ISVALIDREF(rResult) 
	THEN
		MEMCPY(ADR(rResult), ADR(ResultStr), 2 * (MID + 1)); 
	END_IF
ELSE
	IF __ISVALIDREF(rResult) 
	THEN
		MEMMOVE(ADR(rResult), ADR(rStr), 2 * (str1Len + 1)); 
	END_IF
	MID														:= str1Len;
END_IF
END_METHOD

//REPLACE replaces a partial wstring from a larger wstring with a third wstring. REPLACE(STR1, STR2, L, P) 
//means: Replace LEN characters from STR1 with STR2 beginning with the character in the position POS.
METHOD PUBLIC REPLACE : UDINT
VAR_INPUT
	 rSTR1													:	REFERENCE TO T_EXT_WSTRING;
	 STR2													:	T_EXT_WSTRING;
	 LEN													:	UDINT (0..MAX_LENGTH);
	 POS													:	UDINT (0..MAX_LENGTH);
	 rResult												:	REFERENCE TO T_EXT_WSTRING;
END_VAR
VAR
END_VAR
MEMSET(ADR(ResultStr),0,SIZEOF(ResultStr));
IF __ISVALIDREF(rSTR1) 
THEN	
	str1Len 												:= THIS^.LENGTH(rSTR1);
	str2Len 												:= THIS^.LENGTH(STR2);
	
	Pos														:= LIMIT(0,Pos -1, Str1Len);
	Len														:= LIMIT(0,Len,str1Len);
	MEMCPY(ADR(ResultStr), ADR(rSTR1), 2 * Pos); //Copy first part of string 
	MEMCPY(ADR(ResultStr) + (2 * Pos) , ADR(STR2), 2 * (MIN(str2Len + 1, MAX_LENGTH - Pos ))); //insert string two
 	cpyLenght 												:= MAX(0,MIN(str1Len - Pos - Len, MAX_LENGTH - str2Len - Pos));
	MEMCPY(ADR(ResultStr) + (2 * (Pos + str2Len)), ADR(rSTR1) + (2 * (Pos + Len)), 2 * SEL(cpyLenght > 1, 0,cpyLenght));	//Add rest if string 1
	REPLACE 												:= MIN(MAX_LENGTH, Str2Len + pos + MAX(0,Str1Len - Len - Pos));
	IF __ISVALIDREF(rResult) 
	THEN
		MEMMOVE(ADR(rResult), ADR(ResultStr), 2 * (REPLACE + 1)); 
	END_IF	
ELSE
	REPLACE 												:= 0;
END_IF
END_METHOD

//Right returns the right, initial string for a given wstring. RIGHT (STR, SIZE) 
//means: Take the first SIZE character from the right in the string STR.
METHOD PUBLIC RIGHT : UDINT
VAR_INPUT
	 rSTR													: REFERENCE TO WSTRING(MAX_LENGTH);
	 SIZE													: UDINT (0..MAX_LENGTH);
	 rResult												: REFERENCE TO WSTRING(MAX_LENGTH);
END_VAR
VAR
	 chkSize												: UDINT;
END_VAR
MEMSET(ADR(ResultStr),0,SIZEOF(ResultStr));
IF __ISVALIDREF(rSTR)
THEN
	str1Len 												:= LENGTH(rSTR);
	chkSize 												:= MIN(str1Len,MIN(MAX_LENGTH, SIZE));
	MEMCPY(ADR(ResultStr), ADR(rSTR) + (2 * (str1Len - chkSize)), 2* ( chkSize + 1));
	RIGHT													:= chkSize;
	IF __ISVALIDREF(rResult) 
	THEN
		MEMCPY(ADR(rResult), ADR(ResultStr), 2 * (RIGHT + 1)); 
	END_IF	
ELSE
	RIGHT													:= 0;
END_IF
END_METHOD

END_FUNCTION_BLOCK

// ---- POUs/StringHelper/WINSERT_EXT.TcPOU
{attribute 'no_check' := ''}
FUNCTION WINSERT_EXT : WSTRING //The function WINSERT_EXT inserts WSTR2 into WSTR1 at every ITERATION_POSs position  
VAR_INPUT
	STR1													:WSTRING; //Base string - Hint! The base string will cut off if iteration of insertions exceeded the size of the string variable 
	STR2													:WSTRING; //Insert string 
	ITERATION_POS											: INT; //Insert iteration position 
END_VAR
VAR
	Length1,length2,i,iEnd									: INT;														
END_VAR

WINSERT_EXT													:= STR1;
Length1														:= WLEN(STR1);
Length2														:= WLEN(STR2);
IF TO_UINT(Length1 + Length2) > SIZEOF(STR1)
	OR ITERATION_POS = 0
THEN
	;
ELSE
	iEnd													:= ABS(Length1 / ITERATION_POS) - 1;
	FOR i := 1 TO iEnd
	DO 
		WINSERT_EXT											:= WINSERT(WINSERT_EXT,STR2,Length1 - ITERATION_POS * i);
	END_FOR
END_IF

END_FUNCTION

// ---- POUs/System/SystemPulses.TcPOU
{attribute 'no_check'}
//Provides various puslse signals as default
FUNCTION_BLOCK SystemPulses
VAR_INPUT
{attribute 'displaymode':='binary'}
	Options													:	WORD := 2#0000_0001_1110_1110; //Set bit in Options word to enable ot disable existing pulse instances
	PT_ON_Custom											:	TIME := T#30S;	
	PT_OFF_Custom											:	TIME := T#30S;
END_VAR
VAR_OUTPUT
	BlinkSlow												: 	BOOL;
	Blink													: 	BOOL;
	BlinkFast												: 	BOOL;
	BlinkVeryFast											:	BOOL;
	BlinkFlash												:	BOOL;
	
	_20ms													: 	Pulse := (IN := TRUE,	PT_OFF := T#20MS, 		PT_ON := T#20MS);	//20ms						Options .0
	_100ms													: 	Pulse := (IN := TRUE,	PT_OFF := T#100MS, 		PT_ON := T#100MS); 	//10Hz (0.1s) pulse			Options .1
	_250ms													: 	Pulse := (IN := TRUE,	PT_OFF := T#250MS, 		PT_ON := T#250MS); 	//4 Hz - Blink very Fast	Options .2
	_400ms													: 	Pulse := (IN := TRUE,	PT_OFF := T#400MS, 		PT_ON := T#400MS); 	//2.5Hz - Blink Fast *)		Options .3
	_500ms													: 	Pulse := (IN := TRUE,	PT_OFF := T#500MS, 		PT_ON := T#500MS); 	//2Hz / 500ms				Options .4
	_800ms													: 	Pulse := (IN := TRUE,	PT_OFF := T#800MS, 		PT_ON := T#800MS); 	//1.25Hz - Blink normal 	Options .5
	_1s														: 	Pulse := (IN := TRUE,	PT_OFF := T#1S, 		PT_ON := T#1S); 	//1Hz /1s					Options .6
	_1s600ms												: 	Pulse := (IN := TRUE,	PT_OFF := T#1S600MS, 	PT_ON := T#1S600MS);//0.625Hz - Blink slow 		Options .7
	_2s														: 	Pulse := (IN := TRUE,	PT_OFF := T#2S, 		PT_ON := T#2S); 	//0.5Hz						Options .8
	_5s														: 	Pulse := (IN := TRUE,	PT_OFF := T#5S, 		PT_ON := T#5S); 	//5s						Options .9
	_10s													: 	Pulse := (IN := TRUE, 	PT_OFF := T#10S, 		PT_ON := T#10S); 	//10s						Options .10
	_1m														: 	Pulse := (IN := TRUE, 	PT_OFF := T#1M, 		PT_ON := T#1M); 	//1m						Options .11	
	_5m														: 	Pulse := (IN := TRUE, 	PT_OFF := T#5M, 		PT_ON := T#5M); 	//5m						Options .12
	_10m													: 	Pulse := (IN := TRUE, 	PT_OFF := T#10M, 		PT_ON := T#10M); 	//10m						Options .13
	_60m													: 	Pulse := (IN := TRUE, 	PT_OFF := T#60M, 		PT_ON := T#60M); 	//60m						Options .14
	_Custom													: 	Pulse := (IN := TRUE, 	PT_OFF := T#30S, 		PT_ON := T#60M); 	//60m						Options .15
	_Flash													: 	Pulse := (IN := TRUE, 	PT_OFF := T#800MS, 		PT_ON := T#80MS);	//800ms/80ms Blink as flash light
END_VAR                                                            
VAR                                                                
END_VAR

(************************************************************************************************************)
(* function-block generates different pulse signals															*)
(************************************************************************************************************)

(* impuls generator *****************************************************************************************)
_Flash(Q => BlinkFlash); 
IF Options.0 THEN _20ms(Q => ); 				END_IF
IF Options.1 THEN _100ms(Q => ); 				END_IF
IF Options.2 THEN _250ms(Q => BlinkVeryFast); 	END_IF
IF Options.3 THEN _400ms(Q => BlinkFast); 		END_IF
IF Options.4 THEN _500ms(Q => ); 				END_IF
IF Options.5 THEN _800ms(Q => Blink); 			END_IF
IF Options.6 THEN _1s(Q => ); 					END_IF
IF Options.7 THEN _1s600ms(Q => BlinkSlow); 	END_IF
IF Options.8 THEN _2s(Q => ); 					END_IF
IF Options.9 THEN _5s(Q => ); 					END_IF
IF Options.10 THEN _10s(Q => ); 				END_IF
IF Options.11 THEN _1m(Q => ); 					END_IF
IF Options.12 THEN _5m(Q => ); 					END_IF
IF Options.13 THEN _10m(Q => ); 				END_IF
IF Options.14 THEN _60m(Q => ); 				END_IF
IF Options.15 THEN _Custom(PT_OFF := PT_OFF_Custom, PT_ON := PT_ON_Custom ,Q => );	END_IF

(************************************************************************************************)

PROPERTY PUBLIC optAllOn : bool
GET
optAllOn := OPtions = 2#1111_1111_1111_1111;
END_GET
SET
If optAllOn then OPtions := 2#1111_1111_1111_1111; End_if
END_SET
END_PROPERTY

PROPERTY PUBLIC optEnable100ms : bool
GET
optEnable100ms := Options.0;
END_GET
SET
Options.0 := optEnable100ms;
END_SET
END_PROPERTY

PROPERTY PUBLIC optEnable10m : bool
GET
optEnable10m := Options.13;
END_GET
SET
Options.13 := optEnable10m;
END_SET
END_PROPERTY

PROPERTY PUBLIC optEnable10s : bool
GET
optEnable10s := Options.10;
END_GET
SET
Options.10 := optEnable10s;
END_SET
END_PROPERTY

PROPERTY PUBLIC optEnable1m : bool
GET
optEnable1m := Options.11;
END_GET
SET
Options.11 := optEnable1m;
END_SET
END_PROPERTY

PROPERTY PUBLIC optEnable1s : bool
GET
optEnable1s := Options.6;
END_GET
SET
Options.6 := optEnable1s;
END_SET
END_PROPERTY

PROPERTY PUBLIC optEnable1s600msBlinkSlow : bool
GET
optEnable1s600msBlinkSlow := Options.7;
END_GET
SET
Options.7 := optEnable1s600msBlinkSlow;
END_SET
END_PROPERTY

PROPERTY PUBLIC optEnable20ms : bool
GET
optEnable20ms := Options.0;
END_GET
SET
Options.0 := optEnable20ms;
END_SET
END_PROPERTY

PROPERTY PUBLIC optEnable250msBlinkVeryFast : bool
GET
optEnable250msBlinkVeryFast := Options.2;
END_GET
SET
Options.2 := optEnable250msBlinkVeryFast;
END_SET
END_PROPERTY

PROPERTY PUBLIC optEnable2s : bool
GET
optEnable2s := Options.8;
END_GET
SET
Options.8 := optEnable2s;
END_SET
END_PROPERTY

PROPERTY PUBLIC optEnable400msBlinkFast : bool
GET
optEnable400msBlinkFast := Options.3;
END_GET
SET
Options.3 := optEnable400msBlinkFast;
END_SET
END_PROPERTY

PROPERTY PUBLIC optEnable500ms : bool
GET
optEnable500ms := Options.4;
END_GET
SET
Options.4 := optEnable500ms;
END_SET
END_PROPERTY

PROPERTY PUBLIC optEnable5m : bool
GET
optEnable5m := Options.12;
END_GET
SET
Options.12 := optEnable5m;
END_SET
END_PROPERTY

PROPERTY PUBLIC optEnable5s : bool
GET
optEnable5s := Options.9;
END_GET
SET
Options.9 := optEnable5s;
END_SET
END_PROPERTY

PROPERTY PUBLIC optEnable60m : bool
GET
optEnable60m := Options.14;
END_GET
SET
Options.14 := optEnable60m;
END_SET
END_PROPERTY

PROPERTY PUBLIC optEnable800msBlink : bool
GET
optEnable800msBlink := Options.5;
END_GET
SET
Options.5 := optEnable800msBlink;
END_SET
END_PROPERTY

PROPERTY PUBLIC optEnableCustom : bool
GET
optEnableCustom:= Options.15;
END_GET
SET
Options.15 := optEnableCustom;
END_SET
END_PROPERTY

END_FUNCTION_BLOCK

// ---- POUs/System/TaskInfo.TcPOU
{attribute 'no_check'}
//Provides all information of PlcTaskSystemInfo corresponding to the caller task of the instance 
FUNCTION_BLOCK TaskInfo
VAR_INPUT
END_VAR
VAR_OUTPUT
	Index													:	INT := 0;
	TaskName          										: 	STRING(63);
	ObjId             										: 	OTCID;
	CycleTime         										: 	UDINT;
	CycleTimeT       										: 	TIME;
	CycleTimeLT       										: 	LTIME;
	CycleTimeFloat											:	LREAL;	
	Priority          										: 	UINT;
	AdsPort           										: 	UINT;
	CycleCount        										: 	UDINT;
	Tasktime												:	ULINT;
	DcTaskTime        										: 	T_DCTIME64;
	LastExecTime      										: 	UDINT; 
	LastExecTimeNS      									: 	UDINT; //Converted in ns 
	LastExecTimeLT      									: 	LTIME; 
	MaxExecTimeLT											:	LTIME;
	FirstCycle        										: 	BOOL;
	CycleTimeExceeded 										: 	BOOL;	
	CycleTimeExceededCount 									: 	UDINT; //Set to 0 via method resetCylceTimeExceeded()
	CycleTimeExceededCountTotal 							: 	UDINT; //Overall count cycle time exeeded
	InCallAfterOutputUpdate									:	BOOL;
	RTViolation												:	BOOL;
END_VAR

VAR
	GETCURTASKINDEX											: 	GETCURTASKINDEX;
	GETTASKTIME												:	GETTASKTIME;
	TaskInterlock											:	BOOL;
END_VAR

	(*	evaluate PlcTaskInfo arrays													*)
	(********************************************************************************)

(* read task info array of caller task ************************************************************************)
	IF GETCURTASKINDEX.index = 0 	
	THEN 
		GETCURTASKINDEX(index => index); 
		//Init
		TaskName          									:= TwinCAT_SystemInfoVarList._TaskInfo[index].TaskName;
		ObjId             									:= TwinCAT_SystemInfoVarList._TaskInfo[index].ObjId;
		CycleTime         									:= TwinCAT_SystemInfoVarList._TaskInfo[index].CycleTime;
		Priority          									:= TwinCAT_SystemInfoVarList._TaskInfo[index].Priority;
		AdsPort           									:= TwinCAT_SystemInfoVarList._TaskInfo[index].AdsPort;
		CycleTimeT											:= LREAL_TO_TIME(UDINT_TO_LREAL(CycleTime) * 0.0001 );
		CycleTimeLT											:= TO_LTIME(CycleTime * 100);
		CycleTimeFloat										:= (UDINT_TO_LREAL(CycleTime) * 0.0001 / 1000.0);		
	END_IF

	//Cylic 
	CycleCount        										:= TwinCAT_SystemInfoVarList._TaskInfo[index].CycleCount;
	DcTaskTime        										:= TO_ULINT(TwinCAT_SystemInfoVarList._TaskInfo[index].DcTaskTime); 
	LastExecTime      										:= TwinCAT_SystemInfoVarList._TaskInfo[index].LastExecTime; 
	LastExecTimeNS											:= TwinCAT_SystemInfoVarList._TaskInfo[index].LastExecTime * 100;
	LastExecTimeLT      									:= TO_LTIME(LastExecTimeNS); //Converted into ns 
	MaxExecTimeLT											:= MAX(LastExecTimeLT,MaxExecTimeLT);
	
	FirstCycle        										:= TwinCAT_SystemInfoVarList._TaskInfo[index].FirstCycle;
	CycleTimeExceeded 										:= TwinCAT_SystemInfoVarList._TaskInfo[index].CycleTimeExceeded;
	IF CycleTimeExceeded 
	THEN
		CycleTimeExceededCount								:= CycleTimeExceededCount + 1;	
		CycleTimeExceededCountTotal							:= CycleTimeExceededCountTotal + 1;
	END_IF
	InCallAfterOutputUpdate									:= TwinCAT_SystemInfoVarList._TaskInfo[index].InCallAfterOutputUpdate;
	RTViolation												:= TwinCAT_SystemInfoVarList._TaskInfo[index].RTViolation;
	
	//Read time when task suppose to start
	GETTASKTIME(timeLoDW => Tasktime);	
	MEMCPY(ADR(Tasktime) + SIZEOF(GETTASKTIME.timeHiDW),ADR(GETTASKTIME.timeHiDW),SIZEOF(GETTASKTIME.timeHiDW));
	
(**************************************************************************************************)

